(* Logix 5000 project; controller ABB_Drive_Test vendor 1 type 14 code 151 rev 33.13; software revision 33.01 *)

TASK MainTask (continuous, watchdog 500 ms) : T000_MainProgram

MODULES
   Local : vendor 1 type 14 code 151 (Compact 0, rev 33.13)
      Analog_IO : Embedded (Compact 2, rev 1.1, Output RPI 80 ms)
      Module_Hart : vendor 58 type 10 code 4 (Compact 4, rev 3.1, Output RPI 80 ms)
      Discrete_IO : Embedded (Compact 1, rev 3.1, Output RPI 20 ms)
      Counters : Embedded (Compact 3, rev 1.1, Output RPI 20 ms)
      PLC : 1769-L32E Ethernet Port (Ethernet 192.168.2.131, rev 20.1)
         PLC_Controller : vendor 1 type 14 code 77 (CompactLogixL32EController 0, rev 20.1, $7a3aac4c$ RPI 20 ms, $3ca1aa1f$ RPI 20 ms, $2d7d331d$ RPI 20 ms)
      ABBDrive : ETHERNET-MODULE (Ethernet 192.168.2.9, rev 1.1, Output RPI 20 ms)
           ABBDrive:I.Data[0]   // Logic Status Word
           ABBDrive:I.Data[1]   // RPM Actual (INT)
           ABBDrive:I.Data[2]   // DL 1 (Real)
           ABBDrive:I.Data[3]   // DL 1 (Real)
END_MODULES

TYPE ABB_Read :   // Datalinks de Lectura
STRUCT
   Logic_Status_Word : LSW;
   RPM_Feedback : INT;   // RPM Tomada del VSD
   RPM_Referencia : INT;   // Referencia RPM Inyectada
   Output_Power : REAL;
   BusDC : REAL;
   Output_Current : REAL;
   Output_Voltage : REAL;
   PF : REAL;   // Factor de Potencia
   Latest_Fault : INT;
   Accel : BOOL;   // Estado VSD si esta Acelerando
   Descell : BOOL;   // Estado VSD si esta Deshacelerando
END_STRUCT
END_TYPE

TYPE ABB_Write :
STRUCT
   RPM_Reference : INT;
   Run_Forward : BOOL;
   Run_Reverse : BOOL;
   Reset_Fault : BOOL;
END_STRUCT
END_TYPE

TYPE ComandVSD :   // Comandos de funcionamiento VSD
STRUCT
   start : BOOL;   // arranque
   stop : BOOL;   // Parada
   reset : BOOL;   // reset VSD
   referencia : REAL;   // Referencia en RPM para VSD AFE
   direction : BOOL;   // Fordware o Reverse
END_STRUCT
END_TYPE

TYPE Dinagrama :   // Estructura para el dinagrama
STRUCT
   vPotencia : REAL[500];   // captura del vector de potencia
   vCarga : REAL[500];   // captura del vector de carga
   vPosicion : REAL[500];   // captura del vector posicion
   vProximetro : DINT[500];   // captura del vector del proximetro
   NumeroMuestras : INT;
   enabled : BOOL;
   captura : BOOL;   // Flag que indica la captura del sistema
   resetVector : BOOL;   // Flag para darle Reset al vector de posición y carga
   vEmptyREAL : REAL[500];
   vEmptyINT : DINT[500];
   tMuestreo : REAL;   // Tiempo de Muestreo de captura
END_STRUCT
END_TYPE

TYPE ethImplicitRead :   // Comunicación para la lectura de los parametros del VSD por ethernet IP
STRUCT
   Enabled : BOOL;   // habilitar Comunicación
   Done : BOOL;   // Se realizó correctamente
   Error : BOOL;   // Se tiene un error en la lectura de los parámetros
   Value : DINT;   // Valor Obtenido
   instance : DINT;   // instancia del parametro
   atribute : INT;   // Atributo del parametro
END_STRUCT
END_TYPE

TYPE ethImplicitWrite :   // Comunicación Para enviar parametros al sistema
STRUCT
   Enabled : BOOL;   // Habilitar
   Done : BOOL;   // Se realizo exitozamente
   ERR : BOOL;   // Error en el envio de la información
   Value : DINT;   // Valor a ingresar
   Instance : DINT;   // Valor de la Instancia
   Atribute : INT;   // Valor del Atributo de la instancia
   clase : INT;
END_STRUCT
END_TYPE

TYPE fuenteEntradaAnaloga :   // Definición de Entrada Analoga ,Fuente de la señal ,rango minimo y maximo
STRUCT
   fuente : INT;   // Canal por el cual se suministra la señal
   Valor : REAL;   // Valor Actual de la señal
   min : REAL;
   max : REAL;
   ValorMinAmp : REAL;
END_STRUCT
END_TYPE

TYPE LSW :   // Drive - Logic Status Word
STRUCT
   Faulted : BOOL;
   Warning : BOOL;
   RunForward : BOOL;
   RunReverse : BOOL;
   Ready : BOOL;
   RemoteRef : BOOL;
   RemoteCrtl : BOOL;
   AtSpeed : BOOL;
END_STRUCT
END_TYPE

TYPE SWC :   // Comunicación Ethernet con el SWC PRO
STRUCT
   comand : ComandVSD;   // Comandos para VSD
   Dinagrama : Dinagrama;   // Valores para adquisión del dinagrama
   entradasDigitales : INT;
   salidasDigitales : INT;
   entradasAnalogas : REAL[4];
   salidasAnalogas : REAL[4];
   ABBRead : ABB_Read;   // Valores de Lectura
   etheWrite : ethImplicitWrite;   // Valores de Escritura Ethernet para VSD
   etheRead : ethImplicitRead;   // Valores de Lectura
END_STRUCT
END_TYPE

VAR_GLOBAL   (* controller tags *)
   ABB_GetAtt_Value : DINT := 6000;
   ABB_GetMsg : MESSAGE;
        MessageParameters(ServiceCode := 16#000e, DestinationTag := ABB_GetAtt_Value, ...)
   ABB_Input : ABB_Read := (Logic_Status_Word.Ready := 1, Logic_Status_Word.RemoteRef := 1, Logic_Status_Word.RemoteCrtl := 1, RPM_Referencia := 72, Output_Power := 5.960401e-37, BusDC := 715.4, PF := 1.0, Latest_Fault := 28801);
   ABB_Msg_SetValue : DINT := 1;
   ABB_Output : ABB_Write := (RPM_Reference := 72);
   ABB_SetMsg : MESSAGE;
        MessageParameters(ServiceCode := 16#0010, LocalElement := ABB_Msg_SetValue, ...)
   counters : COUNTER[20];
        [0]   // C indice Dinagrama
   Proximetro : BOOL;
   SRP_Displacement_Actual : REAL := 11.377348;
   SRP_Load_Actual : REAL := 10.545264;
   SRP_SimActualStroke : DINT;
   SWC : SWC := (comand.referencia := 72.0, comand.direction := 1, Dinagrama.tMuestreo := 0.05, entradasAnalogas[0] := 16.901644, entradasAnalogas[1] := 13.587194, entradasAnalogas[2] := 3.2056525, entradasAnalogas[3] := 3.2056525, ABBRead.Logic_Status_Word.Ready := 1, ABBRead.Logic_Status_Word.RemoteRef := 1, ABBRead.Logic_Status_Word.RemoteCrtl := 1, ABBRead.RPM_Referencia := 72, ABBRead.Output_Power := 5.960401e-37, ABBRead.BusDC := 714.3, ABBRead.PF := 1.0, ABBRead.Latest_Fault := 28801, etheWrite.Value := 1, etheWrite.Instance := 99, etheWrite.Atribute := 13, etheRead.Value := 6000, etheRead.instance := 99, etheRead.atribute := 7);
   Timmers : TIMER[10] := ([0].PRE := 43, [1].PRE := 828000, [1].ACC := 352537, [1].EN := 1, [1].TT := 1, [2].PRE := 500, [3].PRE := 200, [4].PRE := 10000);
        [0]   // tMuestreo
        [1]   // tPausa
        [2]   // reset del done write ethet
        [3]   // reset del done read eth
        [4]   // reset de la flag de arranque
END_VAR

PROGRAM T000_MainProgram   (* main routine R00_MainRoutine *)
VAR
   Acell : BOOL;
   Captura : BOOL := 1;
   contadorAux : ALIAS FOR counter[0].ACC;
   counter : COUNTER[10] := ([0].DN := 1);
   DesAcell : BOOL;
   Flag : BOOL;
   flagDesAcell : BOOL;   // Flag Auxiliar Boton de Parada
   indiceLocal : DINT;
   InicioDinagram : BOOL := 1;   // Inicio de la Adquisión del Dinagrama
   myoneshot : BOOL[32];
        [0]   // oneshot toogle bot dinagrama
        [2]   // reset de la flag cuando se habilita y se deshabilita
        [1]   // oneshor reset del ocntador
   numeroMuestras : DINT := 640;   // Numero de Muestras del Stroke
   pausa : BOOL := 1;
   Proximetro_Virtual : ALIAS FOR SRP_SimActualStroke;
   rpmFeedback : INT;   // Valor absoluto de la referencia 0 no lo toma
   SCL_01 : SCALE := (In := 16890.0, InRawMax := 19987.0, InRawMin := 3994.0, InEUMax := 20.0, InEUMin := 4.0, Out := 16.901644);
   SCL_02 : SCALE := (In := 13577.0, InRawMax := 19987.0, InRawMin := 3994.0, InEUMax := 20.0, InEUMin := 4.0, Out := 13.587194);
   SCL_03 : SCALE := (In := 3200.0, InRawMax := 19987.0, InRawMin := 3994.0, InEUMax := 20.0, InEUMin := 4.0, Out := 3.2056525, MinAlarm := 1);
   SCL_04 : SCALE := (In := 3200.0, InRawMax := 19987.0, InRawMin := 3994.0, InEUMax := 20.0, InEUMin := 4.0, Out := 3.2056525, MinAlarm := 1);
   SPM_Reference : REAL := 8.5;
   timer : TIMER[10] := ([0].PRE := 50);
        [0]   // Tiempo Muestreo
   VCarga : REAL[1500] := ([0] := 11.827799, [1] := 8.980304, [2] := 8.936409, [3] := 8.84487, [4] := 8.84487, [5] := 8.963797, [6] := 8.963797, [7] := 8.966047, [8] := 8.966047, [9] := 8.860626, [10] := 8.860626, [11] := 9.400863, [12] := 9.400863, [13] := 9.521291, [14] := 9.4916525, [15] := 9.4916525, [16] := 9.597824, [17] := 9.597824, [18] := 9.593322, [19] := 9.593322, [20] := 9.387732, [21] := 9.387732, [22] := 9.403114, [23] := 9.403114, [24] := 9.185143, [25] := 9.185143, [26] := 8.987057, [27] := 8.668918, [28] := 8.668918, [29] := 8.395048, [30] := 8.395048, [31] := 7.648096, [32] := 7.648096, [33] := 7.4162445, [34] := 7.4162445, [35] := 7.2624273, [36] := 7.2624273, [37] := 6.939786, [38] := 6.784468, [39] := 6.784468, [40] := 6.619771, [41] := 6.619771, [42] := 6.1519413, [43] := 6.1519413, [44] := 6.0791597, [45] := 6.0791597, [46] := 6.3091354, [47] := 6.3091354, [48] := 6.480585, [49] := 6.480585, [50] := 6.990058, [51] := 7.45151, [52] := 7.45151, [53] := 7.4702682, [54] := 7.4702682, [55] := 7.577565, [56] := 7.577565, [57] := 7.7895327, [58] := 7.7895327, [59] := 7.948227,
        [60] := 7.948227, [61] := 8.027012, [62] := 8.353029, [63] := 8.353029, [64] := 8.441193, [65] := 8.441193, [66] := 8.438942, [67] := 8.438942, [68] := 8.222097, [69] := 8.222097, [70] := 8.014256, [71] := 8.014256, [72] := 8.062653, [73] := 8.062653, [74] := 8.050648, [75] := 8.092665, [76] := 8.092665, [77] := 8.186457, [78] := 8.186457, [79] := 8.133558, [80] := 8.133558, [81] := 8.182329, [82] := 8.182329, [83] := 8.211593, [84] := 8.211593, [85] := 8.28625, [86] := 8.660664, [87] := 8.660664, [88] := 8.850497, [89] := 8.850497, [90] := 9.020447, [91] := 9.020447, [92] := 9.068843, [93] := 9.068843, [94] := 9.367474, [95] := 9.367474, [96] := 9.479647, [97] := 9.479647, [98] := 9.492778, [99] := 9.546427, [100] := 9.546427, [101] := 9.607578, [102] := 9.607578, [103] := 9.483774, [104] := 9.483774, [105] := 9.460889, [106] := 9.460889, [107] := 9.368223, [108] := 9.368223, [109] := 9.679609, [110] := 10.03639, [111] := 10.03639, [112] := 10.411555, [113] := 10.411555, [114] := 10.760458, [115] := 10.760458, [116] := 10.886138, [117] := 10.886138, [118] := 11.210654, [119] := 11.210654,
        [120] := 11.363346, [121] := 11.575314, [122] := 11.575314, [123] := 11.714874, [124] := 11.714874, [125] := 11.875445, [126] := 11.875445, [127] := 11.921966, [128] := 11.921966, [129] := 11.762521, [130] := 11.762521, [131] := 11.252673, [132] := 11.252673, [133] := 11.074845, [134] := 10.70906, [135] := 10.70906, [136] := 10.527856, [137] := 10.527856, [138] := 10.288126, [139] := 10.288126, [140] := 10.021759, [141] := 10.021759, [142] := 9.853685, [143] := 9.853685, [144] := 9.544551, [145] := 9.442506, [146] := 9.442506, [147] := 9.472519, [148] := 9.472519, [149] := 9.855186, [150] := 9.855186, [151] := 9.900206, [152] := 9.900206, [153] := 10.149315, [154] := 10.149315, [155] := 10.241606, [156] := 10.265241, [157] := 10.265241, [158] := 10.363909, [159] := 10.363909, [160] := 10.395048, [161] := 10.395048, [162] := 10.3444, [163] := 10.3444, [164] := 10.475332, [165] := 10.475332, [166] := 10.469706, [167] := 10.469706, [168] := 10.228475, [169] := 9.813543, [170] := 9.813543, [171] := 9.537798, [172] := 9.537798, [173] := 9.315701, [174] := 9.315701, [175] := 9.132996, [176] := 9.132996, [177] := 9.119114, [178] := 9.119114, [179] := 8.870006,
        [180] := 8.735697, [181] := 8.735697, [182] := 8.758582, [183] := 8.758582, [184] := 8.534609, [185] := 8.534609, [186] := 8.67642, [187] := 8.67642, [188] := 9.151003, [189] := 9.151003, [190] := 9.39336, [191] := 9.39336, [192] := 9.578316, [193] := 9.796661, [194] := 9.796661, [195] := 9.773776, [196] := 9.773776, [197] := 9.757269, [198] := 9.757269, [199] := 9.786156, [200] := 9.786156, [201] := 9.807541, [202] := 9.807541, [203] := 9.934346, [204] := 9.906584, [205] := 9.906584, [206] := 9.544926, [207] := 9.544926, [208] := 9.334833, [209] := 9.334833, [210] := 9.290565, [211] := 9.290565, [212] := 9.1633835, [213] := 9.1633835, [214] := 8.979178, [215] := 9.039205, [216] := 9.039205, [217] := 8.922528, [218] := 8.922528, [219] := 8.92628, [220] := 8.92628, [221] := 8.94879, [222] := 8.94879, [223] := 8.869631, [224] := 8.869631, [225] := 9.230538, [226] := 9.230538, [227] := 9.474395, [228] := 9.451135, [229] := 9.451135, [230] := 9.526167, [231] := 9.526167, [232] := 9.65785, [233] := 9.65785, [234] := 9.437254, [235] := 9.437254, [236] := 9.396736, [237] := 9.396736, [238] := 9.276684, [239] := 9.276684,
        [240] := 9.073344, [241] := 8.794222, [242] := 8.794222, [243] := 8.592009, [244] := 8.592009, [245] := 7.9212155, [246] := 7.9212155, [247] := 7.471769, [248] := 7.471769, [249] := 7.410617, [250] := 7.410617, [251] := 7.0429564, [252] := 6.733821, [253] := 6.733821, [254] := 6.701932, [255] := 6.701932, [256] := 6.272744, [257] := 6.272744, [258] := 6.0765333, [259] := 6.0765333, [260] := 6.197336, [261] := 6.197336, [262] := 6.3331456, [263] := 6.6576624, [264] := 6.6576624, [265] := 6.9412866, [266] := 6.9412866, [267] := 7.467267, [268] := 7.467267, [269] := 7.4646406, [270] := 7.4646406, [271] := 7.641343, [272] := 7.641343, [273] := 7.919339, [274] := 7.919339, [275] := 7.933221, [276] := 8.245732, [277] := 8.245732, [278] := 8.452448, [279] := 8.452448, [280] := 8.443819, [281] := 8.443819, [282] := 8.419058, [283] := 8.419058, [284] := 8.013506, [285] := 8.013506, [286] := 8.006377, [287] := 8.051773, [288] := 8.051773, [289] := 8.016132, [290] := 8.016132, [291] := 8.186081, [292] := 8.186081, [293] := 8.177452, [294] := 8.177452, [295] := 8.110298, [296] := 8.110298, [297] := 8.171075, [298] := 8.210467, [299] := 8.210467,
        [300] := 8.3988, [301] := 8.3988, [302] := 8.589007, [303] := 8.589007, [304] := 8.928906, [305] := 8.928906, [306] := 9.02795, [307] := 9.02795, [308] := 9.220784, [309] := 9.419996, [310] := 9.419996, [311] := 9.439505, [312] := 9.439505, [313] := 9.462765, [314] := 9.462765, [315] := 9.537047, [316] := 9.537047, [317] := 9.573063, [318] := 9.573063, [319] := 9.490152, [320] := 9.4698925, [321] := 9.4698925, [322] := 9.459013, [323] := 9.459013, [324] := 9.643969, [325] := 9.643969, [326] := 10.221722, [327] := 10.221722, [328] := 10.381166, [329] := 10.381166, [330] := 10.706809, [331] := 10.706809, [332] := 11.081974, [333] := 11.236916, [334] := 11.236916, [335] := 11.451885, [336] := 11.451885, [337] := 11.557682, [338] := 11.557682, [339] := 11.815419, [340] := 11.815419, [341] := 11.894579, [342] := 11.894579, [343] := 11.83943, [344] := 11.502533, [345] := 11.502533, [346] := 11.23354, [347] := 11.23354, [348] := 10.874508, [349] := 10.874508, [350] := 10.510599, [351] := 10.510599, [352] := 10.356781, [353] := 10.356781, [354] := 10.096416, [355] := 10.096416, [356] := 9.954229, [357] := 9.64622, [358] := 9.64622, [359] := 9.505158,
        [360] := 9.505158, [361] := 9.400863, [362] := 9.400863, [363] := 9.780153, [364] := 9.780153, [365] := 9.882948, [366] := 9.882948, [367] := 10.071281, [368] := 10.19546, [369] := 10.19546, [370] := 10.254736, [371] := 10.254736, [372] := 10.277621, [373] := 10.277621, [374] := 10.384542, [375] := 10.384542, [376] := 10.339899, [377] := 10.339899, [378] := 10.465578, [379] := 10.506472, [380] := 10.506472, [381] := 10.054024, [382] := 10.054024, [383] := 9.839805, [384] := 9.839805, [385] := 9.606077, [386] := 9.606077, [387] := 9.399737, [388] := 9.399737, [389] := 9.1281185, [390] := 9.1281185, [391] := 9.126243, [392] := 8.908272, [393] := 8.908272, [394] := 8.755205, [395] := 8.755205, [396] := 8.7780905, [397] := 8.7780905, [398] := 8.501595, [399] := 8.501595, [400] := 8.5837555, [401] := 8.5837555, [402] := 9.026824, [403] := 9.205777, [404] := 9.205777, [405] := 9.39636, [406] := 9.39636, [407] := 9.727256, [408] := 9.727256, [409] := 9.79591, [410] := 9.79591, [411] := 9.780529, [412] := 9.780529, [413] := 9.807541, [414] := 9.807541, [415] := 9.803789, [416] := 9.897205, [417] := 9.897205, [418] := 9.930969, [419] := 9.930969,
        [420] := 9.623335, [421] := 9.623335, [422] := 9.400488, [423] := 9.400488, [424] := 9.295442, [425] := 9.295442, [426] := 9.008066, [427] := 8.962296, [428] := 8.962296, [429] := 9.047083, [430] := 9.047083, [431] := 8.975801, [432] := 8.975801, [433] := 8.909022, [434] := 8.909022, [435] := 8.966047, [436] := 8.966047, [437] := 8.890639, [438] := 9.06209, [439] := 9.06209, [440] := 9.338211, [441] := 9.338211, [442] := 9.465767, [443] := 9.465767, [444] := 9.556181, [445] := 9.556181, [446] := 9.638342, [447] := 9.638342, [448] := 9.448133, [449] := 9.448133, [450] := 9.385857, [451] := 9.296942, [452] := 9.296942, [453] := 9.101857, [454] := 9.101857, [455] := 8.818608, [456] := 8.818608, [457] := 8.357906, [458] := 8.357906, [459] := 7.983493, [460] := 7.983493, [461] := 7.4822736, [462] := 7.410617, [463] := 7.410617, [464] := 7.021572, [465] := 7.021572, [466] := 6.8223596, [467] := 6.8223596, [468] := 6.7008066, [469] := 6.7008066, [470] := 6.2479835, [471] := 6.2479835, [472] := 6.0566497, [473] := 6.0566497, [474] := 6.2190957, [475] := 6.393172, [476] := 6.393172, [477] := 6.8107295, [478] := 6.8107295, [479] := 7.374226,
        [480] := 7.374226, [481] := 7.45076, [482] := 7.45076, [483] := 7.5531793, [484] := 7.5531793, [485] := 7.767773, [486] := 7.942975, [487] := 7.942975, [488] := 8.143312, [489] := 8.143312, [490] := 8.344026, [491] := 8.344026, [492] := 8.444944, [493] := 8.444944, [494] := 8.4396925, [495] := 8.4396925, [496] := 8.304258, [497] := 8.096416, [498] := 8.096416, [499] := 8.028888, [500] := 8.028888, [501] := 8.033765, [502] := 8.033765, [503] := 8.07991, [504] := 8.07991, [505] := 8.186457, [506] := 8.186457, [507] := 8.135059, [508] := 8.135059, [509] := 8.197711, [510] := 8.211593, [511] := 8.211593, [512] := 8.229976, [513] := 8.229976, [514] := 8.545488, [515] := 8.545488, [516] := 8.742825, [517] := 8.742825, [518] := 8.9941845, [519] := 8.9941845, [520] := 9.020071, [521] := 9.285313, [522] := 9.285313, [523] := 9.451509, [524] := 9.451509, [525] := 9.517163, [526] := 9.517163, [527] := 9.464266, [528] := 9.464266, [529] := 9.501032, [530] := 9.501032, [531] := 9.53367, [532] := 9.502157, [533] := 9.502157, [534] := 9.4275, [535] := 9.4275, [536] := 9.529919, [537] := 9.529919, [538] := 9.845057, [539] := 9.845057,
        [540] := 10.316263, [541] := 10.316263, [542] := 10.42281, [543] := 10.777716, [544] := 10.777716, [545] := 11.084224, [546] := 11.084224, [547] := 11.248171, [548] := 11.248171, [549] := 11.445131, [550] := 11.445131, [551] := 11.532545, [552] := 11.532545, [553] := 11.782029, [554] := 11.782029, [555] := 11.825172, [556] := 11.940723, [557] := 11.940723, [558] := 11.577189, [559] := 11.577189, [560] := 11.331833, [561] := 11.331833, [562] := 10.911648, [563] := 10.911648, [564] := 10.58338, [565] := 10.58338, [566] := 10.444944, [567] := 10.190208, [568] := 10.190208, [569] := 10.078409, [570] := 10.078409, [571] := 9.809792, [572] := 9.809792, [573] := 9.529544, [574] := 9.529544, [575] := 9.457888, [576] := 9.457888, [577] := 9.594072, [578] := 9.594072, [579] := 9.784656, [580] := 9.956106, [581] := 9.956106, [582] := 10.071656, [583] := 10.071656, [584] := 10.249859, [585] := 10.249859, [586] := 10.2806225, [587] := 10.2806225, [588] := 10.339523, [589] := 10.339523, [590] := 10.348528, [591] := 10.3391485, [592] := 10.3391485, [593] := 10.590883, [594] := 10.590883, [595] := 10.506846, [596] := 10.506846, [597] := 10.029263, [598] := 10.029263, [599] := 9.728756,
        [600] := 9.728756, [601] := 9.62221, [602] := 9.1933975, [603] := 9.1933975, [604] := 9.127743, [605] := 9.127743, [606] := 9.046708, [607] := 9.046708, [608] := 8.771712, [609] := 8.771712, [610] := 8.722941, [611] := 8.722941, [612] := 8.703433, [613] := 8.556744, [614] := 8.556744, [615] := 8.787845, [616] := 8.787845, [617] := 9.044832, [618] := 9.044832, [619] := 9.310448, [620] := 9.310448, [621] := 9.667979, [622] := 9.667979, [623] := 9.759895, [624] := 9.779028, [625] := 9.779028, [626] := 9.782405, [627] := 9.782405, [628] := 9.8082905, [629] := 9.8082905, [630] := 9.803413, [631] := 9.803413, [632] := 9.923091, [633] := 9.923091, [634] := 9.797411, [635] := 9.345714, [636] := 9.345714, [637] := 9.306322, [638] := 9.306322, [639] := 9.172388, [640] := 9.172388, [641] := 11.520915, [642] := 11.266179, [643] := 10.959294, [644] := 10.632902, [645] := 10.337273, [646] := 9.96511, [647] := 9.549427, [648] := 9.102608, [649] := 8.607766, [650] := 8.366911, [651] := 7.9463515, [652] := 7.4500093, [653] := 7.020071, [654] := 6.6572876, [655] := 6.3882947, [656] := 6.1879573, [657] := 6.123429, [658] := 6.1515665, [659] := 6.306509,
        [660] := 6.5207276, [661] := 6.867755, [662] := 7.260176, [663] := 7.6889887, [664] := 8.14819, [665] := 8.538361, [666] := 9.081598, [667] := 9.579441, [668] := 10.054773, [669] := 10.433314, [670] := 10.879759, [671] := 11.271807, [672] := 11.602701, [673] := 11.830425, [674] := 11.960233, [675] := 12.053648, [676] := 12.062277, [677] := 11.9992485, [678] := 11.901332, [679] := 11.737385, [680] := 11.539298, [681] := 11.306321, [682] := 11.069968, [683] := 10.769087, [684] := 10.393923, [685] := 10.046896, [686] := 9.717501, [687] := 9.266179, [688] := 8.839993, [689] := 8.358657, [690] := 7.861564, [691] := 7.5719376, [692] := 7.1783905, [693] := 6.7642093, [694] := 6.470831, [695] := 6.2318516, [696] := 6.1268053, [697] := 6.1283064, [698] := 6.2566123, [699] := 6.5015945, [700] := 6.829488, [701] := 7.2567997, [702] := 7.5719376, [703] := 8.032264, [704] := 8.511349, [705] := 8.931157, [706] := 9.431252, [707] := 9.95348, [708] := 10.449821, [709] := 10.877884, [710] := 11.1885195, [711] := 11.550178, [712] := 11.802288, [713] := 11.975239, [714] := 12.04577, [715] := 12.064903, [716] := 12.011254, [717] := 11.886701, [718] := 11.722754, [719] := 11.55468,
        [720] := 11.320202, [721] := 11.037329, [722] := 10.713187, [723] := 10.439317, [724] := 10.081785, [725] := 9.656725, [726] := 9.211781, [727] := 8.746576, [728] := 8.394298, [729] := 7.8938284, [730] := 7.385481, [731] := 7.0384545, [732] := 6.6576624, [733] := 6.37704, [734] := 6.25061, [735] := 6.135434, [736] := 6.132808, [737] := 6.2322264, [738] := 6.4569497, [739] := 6.781467, [740] := 7.156631, [741] := 7.580191, [742] := 7.9636087, [743] := 8.440818, [744] := 8.94879, [745] := 9.467642, [746] := 9.989495, [747] := 10.374788, [748] := 10.827987, [749] := 11.235415, [750] := 11.583942, [751] := 11.786907, [752] := 11.959857, [753] := 12.050648, [754] := 12.062277, [755] := 12.019883, [756] := 11.9020815, [757] := 11.734009, [758] := 11.524292, [759] := 11.287188, [760] := 11.042206, [761] := 10.725567, [762] := 10.368411, [763] := 9.978615, [764] := 9.63459, [765] := 9.160382, [766] := 8.693303, [767] := 8.187207, [768] := 7.703245, [769] := 7.3678484, [770] := 6.9619207, [771] := 6.610392, [772] := 6.3822923, [773] := 6.1935844, [774] := 6.1204276, [775] := 6.166948, [776] := 6.2453575, [777] := 6.5045958, [778] := 6.717689, [779] := 7.077096,
        [780] := 7.525042, [781] := 7.968111, [782] := 8.438566, [783] := 8.844494, [784] := 9.386982, [785] := 9.897205, [786] := 10.383793, [787] := 10.742825, [788] := 11.151003, [789] := 11.49878, [790] := 11.775652, [791] := 11.959482, [792] := 12.040893, [793] := 12.066403, [794] := 12.021384, [795] := 11.910336, [796] := 11.785781, [797] := 11.588445, [798] := 11.33746, [799] := 11.060964, [800] := 11.060964);
   VPosicion : REAL[1500] := ([0] := 97.12999, [1] := 94.7602, [2] := 93.322075, [3] := 92.56549, [4] := 92.56549, [5] := 91.0961, [6] := 91.0961, [7] := 90.23948, [8] := 90.23948, [9] := 88.451195, [10] := 88.451195, [11] := 86.787964, [12] := 86.787964, [13] := 85.76877, [14] := 83.62408, [15] := 83.62408, [16] := 82.62365, [17] := 82.62365, [18] := 80.466446, [19] := 80.466446, [20] := 78.15294, [21] := 78.15294, [22] := 76.933655, [23] := 76.933655, [24] := 74.39504, [25] := 74.39504, [26] := 73.175766, [27] := 70.61214, [28] := 70.61214, [29] := 69.317825, [30] := 69.317825, [31] := 66.622894, [32] := 66.622894, [33] := 63.784153, [34] := 63.784153, [35] := 62.489838, [36] := 62.489838, [37] := 59.6636, [38] := 58.469326, [39] := 58.469326, [40] := 55.436752, [41] := 55.436752, [42] := 52.37916, [43] := 52.37916, [44] := 50.815983, [45] := 50.815983, [46] := 47.683357, [47] := 47.683357, [48] := 46.12018, [49] := 46.12018, [50] := 42.912518, [51] := 39.686108, [52] := 39.686108, [53] := 38.079155, [54] := 38.079155, [55] := 33.921085, [56] := 33.921085, [57] := 32.795597, [58] := 32.795597, [59] := 30.0569,
        [60] := 30.0569, [61] := 26.43031, [62] := 25.311077, [63] := 25.311077, [64] := 22.603638, [65] := 22.603638, [66] := 20.752829, [67] := 20.752829, [68] := 18.23923, [69] := 18.23923, [70] := 16.82611, [71] := 16.82611, [72] := 14.187455, [73] := 14.187455, [74] := 11.79266, [75] := 10.367036, [76] := 10.367036, [77] := 8.122304, [78] := 8.122304, [79] := 6.3465266, [80] := 6.3465266, [81] := 5.589944, [82] := 5.589944, [83] := 4.3706627, [84] := 4.3706627, [85] := 3.826675, [86] := 2.901268, [87] := 2.901268, [88] := 2.5573702, [89] := 2.5573702, [90] := 2.1071732, [91] := 2.1071732, [92] := 2.0008743, [93] := 2.0008743, [94] := 2.0008743, [95] := 2.0008743, [96] := 2.4073033, [97] := 2.4073033, [98] := 2.6949286, [99] := 3.532797, [100] := 3.532797, [101] := 4.0892897, [102] := 4.0892897, [103] := 5.277309, [104] := 5.277309, [105] := 6.9655476, [106] := 6.9655476, [107] := 7.9159617, [108] := 7.9159617, [109] := 9.666729, [110] := 10.861, [111] := 10.861, [112] := 13.07447, [113] := 13.07447, [114] := 15.544301, [115] := 15.544301, [116] := 16.813606, [117] := 16.813606, [118] := 19.714874, [119] := 19.714874,
        [120] := 22.459826, [121] := 23.829174, [122] := 23.829174, [123] := 26.699179, [124] := 26.699179, [125] := 28.068531, [126] := 28.068531, [127] := 31.263674, [128] := 31.263674, [129] := 32.514225, [130] := 32.514225, [131] := 35.302944, [132] := 35.302944, [133] := 38.954544, [134] := 40.624023, [135] := 40.624023, [136] := 43.6566, [137] := 43.6566, [138] := 45.588696, [139] := 45.588696, [140] := 49.415367, [141] := 49.415367, [142] := 51.247417, [143] := 51.247417, [144] := 54.798973, [145] := 57.769024, [146] := 57.769024, [147] := 59.476017, [148] := 59.476017, [149] := 63.05258, [150] := 63.05258, [151] := 66.10392, [152] := 66.10392, [153] := 67.83593, [154] := 67.83593, [155] := 71.32495, [156] := 72.938156, [157] := 72.938156, [158] := 76.15831, [159] := 76.15831, [160] := 77.32133, [161] := 77.32133, [162] := 79.92871, [163] := 79.92871, [164] := 82.8675, [165] := 82.8675, [166] := 84.33064, [167] := 84.33064, [168] := 86.79422, [169] := 87.750885, [170] := 87.750885, [171] := 90.14568, [172] := 90.14568, [173] := 91.15238, [174] := 91.15238, [175] := 93.28456, [176] := 93.28456, [177] := 94.95404, [178] := 94.95404, [179] := 95.823166,
        [180] := 97.292564, [181] := 97.292564, [182] := 97.93659, [183] := 97.93659, [184] := 99.10586, [185] := 99.10586, [186] := 99.98748, [187] := 99.98748, [188] := 100.35015, [189] := 100.35015, [190] := 100.831604, [191] := 100.831604, [192] := 101.10673, [193] := 101.1505, [194] := 101.1505, [195] := 101.07547, [196] := 101.07547, [197] := 100.981674, [198] := 100.981674, [199] := 100.66904, [200] := 100.66904, [201] := 100.43769, [202] := 100.43769, [203] := 99.80617, [204] := 99.11211, [205] := 99.11211, [206] := 98.79322, [207] := 98.79322, [208] := 97.78027, [209] := 97.78027, [210] := 97.2613, [211] := 97.2613, [212] := 96.16706, [213] := 96.16706, [214] := 95.5293, [215] := 94.08491, [216] := 94.08491, [217] := 92.65304, [218] := 92.65304, [219] := 91.77765, [220] := 91.77765, [221] := 90.38329, [222] := 90.38329, [223] := 88.33864, [224] := 88.33864, [225] := 87.469505, [226] := 87.469505, [227] := 85.599945, [228] := 84.59325, [229] := 84.59325, [230] := 82.56111, [231] := 82.56111, [232] := 81.46689, [233] := 81.46689, [234] := 79.20339, [235] := 79.20339, [236] := 76.72732, [237] := 76.72732, [238] := 75.73938, [239] := 75.73938,
        [240] := 73.12574, [241] := 71.85643, [242] := 71.85643, [243] := 69.22404, [244] := 69.22404, [245] := 67.92346, [246] := 67.92346, [247] := 65.19727, [248] := 65.19727, [249] := 62.63365, [250] := 62.63365, [251] := 61.23929, [252] := 58.519352, [253] := 58.519352, [254] := 55.29294, [255] := 55.29294, [256] := 53.81729, [257] := 53.81729, [258] := 50.60339, [259] := 50.60339, [260] := 49.040203, [261] := 49.040203, [262] := 46.74545, [263] := 43.431496, [264] := 43.431496, [265] := 41.937096, [266] := 41.937096, [267] := 38.37304, [268] := 38.37304, [269] := 36.722313, [270] := 36.722313, [271] := 33.46464, [272] := 33.46464, [273] := 31.776405, [274] := 31.776405, [275] := 28.518724, [276] := 26.223969, [277] := 26.223969, [278] := 24.592007, [279] := 24.592007, [280] := 21.57819, [281] := 21.57819, [282] := 18.733194, [283] := 18.733194, [284] := 17.001188, [285] := 17.001188, [286] := 14.350027, [287] := 13.080722, [288] := 13.080722, [289] := 10.773462, [290] := 10.773462, [291] := 9.879321, [292] := 9.879321, [293] := 7.965985, [294] := 7.965985, [295] := 6.3340216, [296] := 6.3340216, [297] := 5.5149136, [298] := 4.2268486, [299] := 4.2268486,
        [300] := 3.61408, [301] := 3.61408, [302] := 2.794972, [303] := 2.794972, [304] := 2.4760842, [305] := 2.4760842, [306] := 2.0634027, [307] := 2.0634027, [308] := 2.0008743, [309] := 2.0008743, [310] := 2.0008743, [311] := 2.4823368, [312] := 2.4823368, [313] := 3.2764344, [314] := 3.2764344, [315] := 3.695366, [316] := 3.695366, [317] := 4.945913, [318] := 4.945913, [319] := 5.6649776, [320] := 7.353216, [321] := 7.353216, [322] := 8.309886, [323] := 8.309886, [324] := 10.235727, [325] := 10.235727, [326] := 12.668043, [327] := 12.668043, [328] := 13.837301, [329] := 13.837301, [330] := 16.150814, [331] := 16.150814, [332] := 17.632713, [333] := 20.171326, [334] := 20.171326, [335] := 23.010067, [336] := 23.010067, [337] := 24.373161, [338] := 24.373161, [339] := 27.918465, [340] := 27.918465, [341] := 29.437876, [342] := 29.437876, [343] := 31.763899, [344] := 35.27168, [345] := 35.27168, [346] := 36.853622, [347] := 36.853622, [348] := 40.08629, [349] := 40.08629, [350] := 41.74951, [351] := 41.74951, [352] := 45.12599, [353] := 45.12599, [354] := 48.658787, [355] := 48.658787, [356] := 50.484585, [357] := 54.173695, [358] := 54.173695, [359] := 55.86194,
        [360] := 55.86194, [361] := 59.288437, [362] := 59.288437, [363] := 61.21428, [364] := 61.21428, [365] := 64.75958, [366] := 64.75958, [367] := 68.28612, [368] := 69.9431, [369] := 69.9431, [370] := 73.182014, [371] := 73.182014, [372] := 74.782715, [373] := 74.782715, [374] := 77.46514, [375] := 77.46514, [376] := 78.796974, [377] := 78.796974, [378] := 81.804535, [379] := 84.64328, [380] := 84.64328, [381] := 85.98762, [382] := 85.98762, [383] := 88.35115, [384] := 88.35115, [385] := 90.24573, [386] := 90.24573, [387] := 91.44626, [388] := 91.44626, [389] := 93.30332, [390] := 93.30332, [391] := 94.00987, [392] := 95.78565, [393] := 95.78565, [394] := 96.529724, [395] := 96.529724, [396] := 97.88657, [397] := 97.88657, [398] := 99.04332, [399] := 99.04332, [400] := 99.46226, [401] := 99.46226, [402] := 100.20634, [403] := 100.51272, [404] := 100.51272, [405] := 100.94416, [406] := 100.94416, [407] := 101.11298, [408] := 101.11298, [409] := 101.13174, [410] := 101.13174, [411] := 101.0317, [412] := 101.0317, [413] := 100.712814, [414] := 100.712814, [415] := 100.45644, [416] := 99.8937, [417] := 99.8937, [418] := 99.599815, [419] := 99.599815,
        [420] := 98.76821, [421] := 98.76821, [422] := 98.31801, [423] := 98.31801, [424] := 97.33007, [425] := 97.33007, [426] := 96.12956, [427] := 95.46051, [428] := 95.46051, [429] := 94.022385, [430] := 94.022385, [431] := 93.34083, [432] := 93.34083, [433] := 91.90271, [434] := 91.90271, [435] := 91.05233, [436] := 91.05233, [437] := 89.21403, [438] := 87.32571, [439] := 87.32571, [440] := 86.38153, [441] := 86.38153, [442] := 84.35565, [443] := 84.35565, [444] := 82.31726, [445] := 82.31726, [446] := 81.26055, [447] := 81.26055, [448] := 79.0846, [449] := 79.0846, [450] := 77.727745, [451] := 75.69561, [452] := 75.69561, [453] := 74.35753, [454] := 74.35753, [455] := 71.89395, [456] := 71.89395, [457] := 69.24279, [458] := 69.24279, [459] := 67.87344, [460] := 67.87344, [461] := 64.98468, [462] := 63.509033, [463] := 63.509033, [464] := 60.98918, [465] := 60.98918, [466] := 59.3197, [467] := 59.3197, [468] := 56.355904, [469] := 56.355904, [470] := 53.31082, [471] := 53.31082, [472] := 51.672607, [473] := 48.32114, [474] := 48.32114, [475] := 46.67667, [476] := 46.67667, [477] := 43.237663, [478] := 43.237663, [479] := 40.498966,
        [480] := 40.498966, [481] := 38.616898, [482] := 38.616898, [483] := 34.971546, [484] := 34.971546, [485] := 32.032764, [486] := 30.382038, [487] := 30.382038, [488] := 27.14312, [489] := 27.14312, [490] := 25.742508, [491] := 25.742508, [492] := 22.341024, [493] := 22.341024, [494] := 20.771587, [495] := 20.771587, [496] := 17.814043, [497] := 15.075344, [498] := 15.075344, [499] := 14.087415, [500] := 14.087415, [501] := 11.830175, [502] := 11.830175, [503] := 10.517102, [504] := 10.517102, [505] := 8.191085, [506] := 8.191085, [507] := 7.434502, [508] := 7.434502, [509] := 5.87132, [510] := 4.564497, [511] := 4.564497, [512] := 3.9454758, [513] := 3.9454758, [514] := 2.9763012, [515] := 2.9763012, [516] := 2.6198955, [517] := 2.6198955, [518] := 2.2072167, [519] := 2.2072167, [520] := 2.0071268, [521] := 2.0008743, [522] := 2.0008743, [523] := 2.1321833, [524] := 2.1321833, [525] := 2.7199388, [526] := 2.7199388, [527] := 3.101358, [528] := 3.101358, [529] := 4.0517716, [530] := 4.0517716, [531] := 4.8708797, [532] := 6.434065, [533] := 6.434065, [534] := 7.2844357, [535] := 7.2844357, [536] := 9.179014, [537] := 9.179014, [538] := 11.217406, [539] := 11.217406,
        [540] := 12.274119, [541] := 12.274119, [542] := 14.837742, [543] := 16.08829, [544] := 16.08829, [545] := 18.389297, [546] := 18.389297, [547] := 19.708622, [548] := 19.708622, [549] := 21.87832, [550] := 21.87832, [551] := 24.779589, [552] := 24.779589, [553] := 26.080154, [554] := 26.080154, [555] := 28.887642, [556] := 30.438316, [557] := 30.438316, [558] := 33.746017, [559] := 33.746017, [560] := 36.62852, [561] := 36.62852, [562] := 38.32927, [563] := 38.32927, [564] := 42.005875, [565] := 42.005875, [566] := 44.663284, [567] := 46.420307, [568] := 46.420307, [569] := 49.94685, [570] := 49.94685, [571] := 51.70387, [572] := 51.70387, [573] := 55.11161, [574] := 55.11161, [575] := 56.631023, [576] := 56.631023, [577] := 60.220093, [578] := 60.220093, [579] := 63.80291, [580] := 65.459885, [581] := 65.459885, [582] := 68.73007, [583] := 68.73007, [584] := 70.38704, [585] := 70.38704, [586] := 73.638466, [587] := 73.638466, [588] := 75.245415, [589] := 75.245415, [590] := 77.99661, [591] := 81.06672, [592] := 81.06672, [593] := 82.42355, [594] := 82.42355, [595] := 84.94341, [596] := 84.94341, [597] := 86.537865, [598] := 86.537865, [599] := 88.65753,
        [600] := 88.65753, [601] := 90.56462, [602] := 91.87144, [603] := 91.87144, [604] := 93.74726, [605] := 93.74726, [606] := 95.46676, [607] := 95.46676, [608] := 96.242096, [609] := 96.242096, [610] := 97.57394, [611] := 97.57394, [612] := 98.1617, [613] := 99.21841, [614] := 99.21841, [615] := 99.67486, [616] := 99.67486, [617] := 100.41892, [618] := 100.41892, [619] := 100.85663, [620] := 100.85663, [621] := 101.01295, [622] := 101.01295, [623] := 101.1505, [624] := 101.11298, [625] := 101.11298, [626] := 100.937904, [627] := 100.937904, [628] := 100.75658, [629] := 100.75658, [630] := 100.30013, [631] := 100.30013, [632] := 99.56231, [633] := 99.56231, [634] := 99.18089, [635] := 98.324265, [636] := 98.324265, [637] := 97.3676, [638] := 97.3676, [639] := 96.829865, [640] := 96.829865, [641] := 92.01525, [642] := 87.76965, [643] := 82.65491, [644] := 77.21503, [645] := 72.28787, [646] := 66.08516, [647] := 59.157127, [648] := 51.71012, [649] := 43.462765, [650] := 39.448513, [651] := 32.43919, [652] := 24.166822, [653] := 17.001188, [654] := 10.954791, [655] := 6.4715805, [656] := 3.1326203, [657] := 2.05715, [658] := 2.5261045, [659] := 5.1084847,
        [660] := 8.678797, [661] := 14.462578, [662] := 21.002937, [663] := 28.149813, [664] := 35.80316, [665] := 42.306007, [666] := 51.35997, [667] := 59.65735, [668] := 67.57956, [669] := 73.88857, [670] := 81.32932, [671] := 87.86345, [672] := 93.37836, [673] := 97.17376, [674] := 99.33721, [675] := 100.89414, [676] := 101.03796, [677] := 99.98748, [678] := 98.35553, [679] := 95.623085, [680] := 92.32163, [681] := 88.43869, [682] := 84.499466, [683] := 79.48477, [684] := 73.23204, [685] := 67.44826, [686] := 61.958355, [687] := 54.436314, [688] := 47.333206, [689] := 39.310944, [690] := 31.026072, [691] := 26.19896, [692] := 19.639843, [693] := 12.736821, [694] := 7.847184, [695] := 3.86419, [696] := 2.1134257, [697] := 2.1384358, [698] := 4.2768717, [699] := 8.359906, [700] := 13.824797, [701] := 20.946663, [702] := 26.19896, [703] := 33.871067, [704] := 41.855812, [705] := 48.852623, [706] := 57.187515, [707] := 65.89133, [708] := 74.1637, [709] := 81.298065, [710] := 86.47533, [711] := 92.50296, [712] := 96.7048, [713] := 99.58732, [714] := 100.76283, [715] := 101.08172, [716] := 100.18758, [717] := 98.11168, [718] := 95.379234, [719] := 92.578,
        [720] := 88.67004, [721] := 83.955475, [722] := 78.553116, [723] := 73.98862, [724] := 68.02976, [725] := 60.945408, [726] := 53.529667, [727] := 45.77627, [728] := 39.904957, [729] := 31.563807, [730] := 23.091352, [731] := 17.307573, [732] := 10.961044, [733] := 6.2839985, [734] := 4.1768284, [735] := 2.257237, [736] := 2.213469, [737] := 3.8704424, [738] := 7.6158314, [739] := 13.024449, [740] := 19.277185, [741] := 26.336521, [742] := 32.726814, [743] := 40.680294, [744] := 49.146496, [745] := 57.794033, [746] := 66.491585, [747] := 72.91315, [748] := 80.466446, [749] := 87.25692, [750] := 93.06571, [751] := 96.44845, [752] := 99.33095, [753] := 100.844124, [754] := 101.03796, [755] := 100.33139, [756] := 98.36803, [757] := 95.56681, [758] := 92.07153, [759] := 88.1198, [760] := 84.03676, [761] := 78.75945, [762] := 72.806854, [763] := 66.31026, [764] := 60.5765, [765] := 52.673042, [766] := 44.88839, [767] := 36.45345, [768] := 28.387415, [769] := 22.797472, [770] := 16.032013, [771] := 10.173202, [772] := 6.3715367, [773] := 3.2264113, [774] := 2.0071268, [775] := 2.782467, [776] := 4.0892897, [777] := 8.409929, [778] := 11.961484, [779] := 17.951601,
        [780] := 25.41737, [781] := 32.80185, [782] := 40.64278, [783] := 47.408234, [784] := 56.44969, [785] := 64.953415, [786] := 73.06321, [787] := 79.04708, [788] := 85.85005, [789] := 91.64634, [790] := 96.26086, [791] := 99.32471, [792] := 100.68154, [793] := 101.10673, [794] := 100.3564, [795] := 98.50559, [796] := 96.42968, [797] := 93.14075, [798] := 88.957664, [799] := 84.349396, [800] := 84.349396);
   VPotencia : REAL[1500] := ([0] := 5.9449345e-37, [1] := 5.9449345e-37, [2] := 5.9449345e-37, [3] := 5.9449345e-37, [4] := 5.9449345e-37, [5] := 5.9449345e-37, [6] := 5.9449345e-37, [7] := 5.9449345e-37, [8] := 5.9449345e-37, [9] := 5.9449345e-37, [10] := 5.9449345e-37, [11] := 5.9449345e-37, [12] := 5.9449345e-37, [13] := 5.9449345e-37, [14] := 5.9449345e-37, [15] := 5.9449345e-37, [16] := 5.9449345e-37, [17] := 5.9449345e-37, [18] := 5.9449345e-37, [19] := 5.9449345e-37, [20] := 5.9449345e-37, [21] := 5.9449345e-37, [22] := 5.9449345e-37, [23] := 5.9449345e-37, [24] := 5.9449345e-37, [25] := 5.9449345e-37, [26] := 5.9449345e-37, [27] := 5.9449345e-37, [28] := 5.9449345e-37, [29] := 5.9449345e-37, [30] := 5.9449345e-37, [31] := 5.9449345e-37, [32] := 5.9449345e-37, [33] := 5.9449345e-37, [34] := 5.9449345e-37, [35] := 5.9449345e-37, [36] := 5.9449345e-37, [37] := 5.9449345e-37, [38] := 5.9449345e-37, [39] := 5.9449345e-37, [40] := 5.9449345e-37, [41] := 5.9449345e-37, [42] := 5.9449345e-37, [43] := 5.9449345e-37, [44] := 5.9449345e-37, [45] := 5.9449345e-37, [46] := 5.9449345e-37, [47] := 5.9449345e-37, [48] := 5.9449345e-37, [49] := 5.9449345e-37, [50] := 5.9449345e-37, [51] := 5.9449345e-37, [52] := 5.9449345e-37, [53] := 5.9449345e-37, [54] := 5.9449345e-37, [55] := 5.9449345e-37, [56] := 5.9449345e-37, [57] := 5.9449345e-37, [58] := 5.9449345e-37, [59] := 5.9449345e-37,
        [60] := 5.9449345e-37, [61] := 5.9449345e-37, [62] := 5.9449345e-37, [63] := 5.9449345e-37, [64] := 5.9449345e-37, [65] := 5.9449345e-37, [66] := 5.9449345e-37, [67] := 5.9449345e-37, [68] := 5.9449345e-37, [69] := 5.9449345e-37, [70] := 5.9449345e-37, [71] := 5.9449345e-37, [72] := 5.9449345e-37, [73] := 5.9449345e-37, [74] := 5.9449345e-37, [75] := 5.9449345e-37, [76] := 5.9449345e-37, [77] := 5.9449345e-37, [78] := 5.9449345e-37, [79] := 5.9449345e-37, [80] := 5.9449345e-37, [81] := 5.9449345e-37, [82] := 5.9449345e-37, [83] := 5.9449345e-37, [84] := 5.9449345e-37, [85] := 5.9449345e-37, [86] := 5.9449345e-37, [87] := 5.9449345e-37, [88] := 5.9449345e-37, [89] := 5.9449345e-37, [90] := 5.9449345e-37, [91] := 5.9449345e-37, [92] := 5.9449345e-37, [93] := 5.9449345e-37, [94] := 5.9449345e-37, [95] := 5.9449345e-37, [96] := 5.9449345e-37, [97] := 5.9449345e-37, [98] := 5.9449345e-37, [99] := 5.9449345e-37, [100] := 5.9449345e-37, [101] := 5.9449345e-37, [102] := 5.9449345e-37, [103] := 5.9449345e-37, [104] := 5.9449345e-37, [105] := 5.9449345e-37, [106] := 5.9449345e-37, [107] := 5.9449345e-37, [108] := 5.9449345e-37, [109] := 5.9449345e-37, [110] := 5.9449345e-37, [111] := 5.9449345e-37, [112] := 5.9449345e-37, [113] := 5.9449345e-37, [114] := 5.9449345e-37, [115] := 5.9449345e-37, [116] := 5.9449345e-37, [117] := 5.9449345e-37, [118] := 5.9449345e-37, [119] := 5.9449345e-37,
        [120] := 5.9449345e-37, [121] := 5.9449345e-37, [122] := 5.9449345e-37, [123] := 5.9449345e-37, [124] := 5.9449345e-37, [125] := 5.9449345e-37, [126] := 5.9449345e-37, [127] := 5.9449345e-37, [128] := 5.9449345e-37, [129] := 5.9449345e-37, [130] := 5.9449345e-37, [131] := 5.9449345e-37, [132] := 5.9449345e-37, [133] := 5.9449345e-37, [134] := 5.9449345e-37, [135] := 5.9449345e-37, [136] := 5.9449345e-37, [137] := 5.9449345e-37, [138] := 5.9449345e-37, [139] := 5.9449345e-37, [140] := 5.9449345e-37, [141] := 5.9449345e-37, [142] := 5.9449345e-37, [143] := 5.9449345e-37, [144] := 5.9449345e-37, [145] := 5.9449345e-37, [146] := 5.9449345e-37, [147] := 5.9449345e-37, [148] := 5.9449345e-37, [149] := 5.9449345e-37, [150] := 5.9449345e-37, [151] := 5.9449345e-37, [152] := 5.9449345e-37, [153] := 5.9449345e-37, [154] := 5.9449345e-37, [155] := 5.9449345e-37, [156] := 5.9449345e-37, [157] := 5.9449345e-37, [158] := 5.9449345e-37, [159] := 5.9449345e-37, [160] := 5.9449345e-37, [161] := 5.9449345e-37, [162] := 5.9449345e-37, [163] := 5.9449345e-37, [164] := 5.9449345e-37, [165] := 5.9449345e-37, [166] := 5.9449345e-37, [167] := 5.9449345e-37, [168] := 5.9449345e-37, [169] := 5.9449345e-37, [170] := 5.9449345e-37, [171] := 5.9449345e-37, [172] := 5.9449345e-37, [173] := 5.9449345e-37, [174] := 5.9449345e-37, [175] := 5.9449345e-37, [176] := 5.9449345e-37, [177] := 5.9449345e-37, [178] := 5.9449345e-37, [179] := 5.9449345e-37,
        [180] := 5.9449345e-37, [181] := 5.9449345e-37, [182] := 5.9449345e-37, [183] := 5.9449345e-37, [184] := 5.9449345e-37, [185] := 5.9449345e-37, [186] := 5.9449345e-37, [187] := 5.9449345e-37, [188] := 5.9449345e-37, [189] := 5.9449345e-37, [190] := 5.9449345e-37, [191] := 5.9449345e-37, [192] := 5.9449345e-37, [193] := 5.9449345e-37, [194] := 5.9449345e-37, [195] := 5.9449345e-37, [196] := 5.9449345e-37, [197] := 5.9449345e-37, [198] := 5.9449345e-37, [199] := 5.9449345e-37, [200] := 5.9449345e-37, [201] := 5.9449345e-37, [202] := 5.9449345e-37, [203] := 5.9449345e-37, [204] := 5.9449345e-37, [205] := 5.9449345e-37, [206] := 5.9449345e-37, [207] := 5.9449345e-37, [208] := 5.9449345e-37, [209] := 5.9449345e-37, [210] := 5.9449345e-37, [211] := 5.9449345e-37, [212] := 5.9449345e-37, [213] := 5.9449345e-37, [214] := 5.9449345e-37, [215] := 5.9449345e-37, [216] := 5.9449345e-37, [217] := 5.9449345e-37, [218] := 5.9449345e-37, [219] := 5.9449345e-37, [220] := 5.9449345e-37, [221] := 5.9449345e-37, [222] := 5.9449345e-37, [223] := 5.9449345e-37, [224] := 5.9449345e-37, [225] := 5.9449345e-37, [226] := 5.9449345e-37, [227] := 5.9449345e-37, [228] := 5.9449345e-37, [229] := 5.9449345e-37, [230] := 5.9449345e-37, [231] := 5.9449345e-37, [232] := 5.9449345e-37, [233] := 5.9449345e-37, [234] := 5.9449345e-37, [235] := 5.9449345e-37, [236] := 5.9449345e-37, [237] := 5.9449345e-37, [238] := 5.9449345e-37, [239] := 5.9449345e-37,
        [240] := 5.9449345e-37, [241] := 5.9449345e-37, [242] := 5.9449345e-37, [243] := 5.9449345e-37, [244] := 5.9449345e-37, [245] := 5.9449345e-37, [246] := 5.9449345e-37, [247] := 5.9449345e-37, [248] := 5.9449345e-37, [249] := 5.9449345e-37, [250] := 5.9449345e-37, [251] := 5.9449345e-37, [252] := 5.9449345e-37, [253] := 5.9449345e-37, [254] := 5.9449345e-37, [255] := 5.9449345e-37, [256] := 5.9449345e-37, [257] := 5.9449345e-37, [258] := 5.9449345e-37, [259] := 5.9449345e-37, [260] := 5.9449345e-37, [261] := 5.9449345e-37, [262] := 5.9449345e-37, [263] := 5.9449345e-37, [264] := 5.9449345e-37, [265] := 5.9449345e-37, [266] := 5.9449345e-37, [267] := 5.9449345e-37, [268] := 5.9449345e-37, [269] := 5.9449345e-37, [270] := 5.9449345e-37, [271] := 5.9449345e-37, [272] := 5.9449345e-37, [273] := 5.9449345e-37, [274] := 5.9449345e-37, [275] := 5.9449345e-37, [276] := 5.9449345e-37, [277] := 5.9449345e-37, [278] := 5.9449345e-37, [279] := 5.9449345e-37, [280] := 5.9449345e-37, [281] := 5.9449345e-37, [282] := 5.9449345e-37, [283] := 5.9449345e-37, [284] := 5.9449345e-37, [285] := 5.9449345e-37, [286] := 5.9449345e-37, [287] := 5.9449345e-37, [288] := 5.9449345e-37, [289] := 5.9449345e-37, [290] := 5.9449345e-37, [291] := 5.9449345e-37, [292] := 5.9449345e-37, [293] := 5.9449345e-37, [294] := 5.9449345e-37, [295] := 5.9449345e-37, [296] := 5.9449345e-37, [297] := 5.9449345e-37, [298] := 5.9449345e-37, [299] := 5.9449345e-37,
        [300] := 5.9449345e-37, [301] := 5.9449345e-37, [302] := 5.9449345e-37, [303] := 5.9449345e-37, [304] := 5.9449345e-37, [305] := 5.9449345e-37, [306] := 5.9449345e-37, [307] := 5.9449345e-37, [308] := 5.9449345e-37, [309] := 5.9449345e-37, [310] := 5.9449345e-37, [311] := 5.9449345e-37, [312] := 5.9449345e-37, [313] := 5.9449345e-37, [314] := 5.9449345e-37, [315] := 5.9449345e-37, [316] := 5.9449345e-37, [317] := 5.9449345e-37, [318] := 5.9449345e-37, [319] := 5.9449345e-37, [320] := 5.9449345e-37, [321] := 5.9449345e-37, [322] := 5.9449345e-37, [323] := 5.9449345e-37, [324] := 5.9449345e-37, [325] := 5.9449345e-37, [326] := 5.9449345e-37, [327] := 5.9449345e-37, [328] := 5.9449345e-37, [329] := 5.9449345e-37, [330] := 5.9449345e-37, [331] := 5.9449345e-37, [332] := 5.9449345e-37, [333] := 5.9449345e-37, [334] := 5.9449345e-37, [335] := 5.9449345e-37, [336] := 5.9449345e-37, [337] := 5.9449345e-37, [338] := 5.9449345e-37, [339] := 5.9449345e-37, [340] := 5.9449345e-37, [341] := 5.9449345e-37, [342] := 5.9449345e-37, [343] := 5.9449345e-37, [344] := 5.9449345e-37, [345] := 5.9449345e-37, [346] := 5.9449345e-37, [347] := 5.9449345e-37, [348] := 5.9449345e-37, [349] := 5.9449345e-37, [350] := 5.9449345e-37, [351] := 5.9449345e-37, [352] := 5.9449345e-37, [353] := 5.9449345e-37, [354] := 5.9449345e-37, [355] := 5.9449345e-37, [356] := 5.9449345e-37, [357] := 5.9449345e-37, [358] := 5.9449345e-37, [359] := 5.9449345e-37,
        [360] := 5.9449345e-37, [361] := 5.9449345e-37, [362] := 5.9449345e-37, [363] := 5.9449345e-37, [364] := 5.9449345e-37, [365] := 5.9449345e-37, [366] := 5.9449345e-37, [367] := 5.9449345e-37, [368] := 5.9449345e-37, [369] := 5.9449345e-37, [370] := 5.9449345e-37, [371] := 5.9449345e-37, [372] := 5.9449345e-37, [373] := 5.9449345e-37, [374] := 5.9449345e-37, [375] := 5.9449345e-37, [376] := 5.9449345e-37, [377] := 5.9449345e-37, [378] := 5.9449345e-37, [379] := 5.9449345e-37, [380] := 5.9449345e-37, [381] := 5.9449345e-37, [382] := 5.9449345e-37, [383] := 5.9449345e-37, [384] := 5.9449345e-37, [385] := 5.9449345e-37, [386] := 5.9449345e-37, [387] := 5.9449345e-37, [388] := 5.9449345e-37, [389] := 5.9449345e-37, [390] := 5.9449345e-37, [391] := 5.9449345e-37, [392] := 5.9449345e-37, [393] := 5.9449345e-37, [394] := 5.9449345e-37, [395] := 5.9449345e-37, [396] := 5.9449345e-37, [397] := 5.9449345e-37, [398] := 5.9449345e-37, [399] := 5.9449345e-37, [400] := 5.9449345e-37, [401] := 5.9449345e-37, [402] := 5.9449345e-37, [403] := 5.9449345e-37, [404] := 5.9449345e-37, [405] := 5.9449345e-37, [406] := 5.9449345e-37, [407] := 5.9449345e-37, [408] := 5.9449345e-37, [409] := 5.9449345e-37, [410] := 5.9449345e-37, [411] := 5.9449345e-37, [412] := 5.9449345e-37, [413] := 5.9449345e-37, [414] := 5.9449345e-37, [415] := 5.9449345e-37, [416] := 5.9449345e-37, [417] := 5.9449345e-37, [418] := 5.9449345e-37, [419] := 5.9449345e-37,
        [420] := 5.9449345e-37, [421] := 5.9449345e-37, [422] := 5.9449345e-37, [423] := 5.9449345e-37, [424] := 5.9449345e-37, [425] := 5.9449345e-37, [426] := 5.9449345e-37, [427] := 5.9449345e-37, [428] := 5.9449345e-37, [429] := 5.9449345e-37, [430] := 5.9449345e-37, [431] := 5.9449345e-37, [432] := 5.9449345e-37, [433] := 5.9449345e-37, [434] := 5.9449345e-37, [435] := 5.9449345e-37, [436] := 5.9449345e-37, [437] := 5.9449345e-37, [438] := 5.9449345e-37, [439] := 5.9449345e-37, [440] := 5.9449345e-37, [441] := 5.9449345e-37, [442] := 5.9449345e-37, [443] := 5.9449345e-37, [444] := 5.9449345e-37, [445] := 5.9449345e-37, [446] := 5.9449345e-37, [447] := 5.9449345e-37, [448] := 5.9449345e-37, [449] := 5.9449345e-37, [450] := 5.9449345e-37, [451] := 5.9449345e-37, [452] := 5.9449345e-37, [453] := 5.9449345e-37, [454] := 5.9449345e-37, [455] := 5.9449345e-37, [456] := 5.9449345e-37, [457] := 5.9449345e-37, [458] := 5.9449345e-37, [459] := 5.9449345e-37, [460] := 5.9449345e-37, [461] := 5.9449345e-37, [462] := 5.9449345e-37, [463] := 5.9449345e-37, [464] := 5.9449345e-37, [465] := 5.9449345e-37, [466] := 5.9449345e-37, [467] := 5.9449345e-37, [468] := 5.9449345e-37, [469] := 5.9449345e-37, [470] := 5.9449345e-37, [471] := 5.9449345e-37, [472] := 5.9449345e-37, [473] := 5.9449345e-37, [474] := 5.9449345e-37, [475] := 5.9449345e-37, [476] := 5.9449345e-37, [477] := 5.9449345e-37, [478] := 5.9449345e-37, [479] := 5.9449345e-37,
        [480] := 5.9449345e-37, [481] := 5.9449345e-37, [482] := 5.9449345e-37, [483] := 5.9449345e-37, [484] := 5.9449345e-37, [485] := 5.9449345e-37, [486] := 5.9449345e-37, [487] := 5.9449345e-37, [488] := 5.9449345e-37, [489] := 5.9449345e-37, [490] := 5.9449345e-37, [491] := 5.9449345e-37, [492] := 5.9449345e-37, [493] := 5.9449345e-37, [494] := 5.9449345e-37, [495] := 5.9449345e-37, [496] := 5.9449345e-37, [497] := 5.9449345e-37, [498] := 5.9449345e-37, [499] := 5.9449345e-37, [500] := 5.9449345e-37, [501] := 5.9449345e-37, [502] := 5.9449345e-37, [503] := 5.9449345e-37, [504] := 5.9449345e-37, [505] := 5.9449345e-37, [506] := 5.9449345e-37, [507] := 5.9449345e-37, [508] := 5.9449345e-37, [509] := 5.9449345e-37, [510] := 5.9449345e-37, [511] := 5.9449345e-37, [512] := 5.9449345e-37, [513] := 5.9449345e-37, [514] := 5.9449345e-37, [515] := 5.9449345e-37, [516] := 5.9449345e-37, [517] := 5.9449345e-37, [518] := 5.9449345e-37, [519] := 5.9449345e-37, [520] := 5.9449345e-37, [521] := 5.9449345e-37, [522] := 5.9449345e-37, [523] := 5.9449345e-37, [524] := 5.9449345e-37, [525] := 5.9449345e-37, [526] := 5.9449345e-37, [527] := 5.9449345e-37, [528] := 5.9449345e-37, [529] := 5.9449345e-37, [530] := 5.9449345e-37, [531] := 5.9449345e-37, [532] := 5.9449345e-37, [533] := 5.9449345e-37, [534] := 5.9449345e-37, [535] := 5.9449345e-37, [536] := 5.9449345e-37, [537] := 5.9449345e-37, [538] := 5.9449345e-37, [539] := 5.9449345e-37,
        [540] := 5.9449345e-37, [541] := 5.9449345e-37, [542] := 5.9449345e-37, [543] := 5.9449345e-37, [544] := 5.9449345e-37, [545] := 5.9449345e-37, [546] := 5.9449345e-37, [547] := 5.9449345e-37, [548] := 5.9449345e-37, [549] := 5.9449345e-37, [550] := 5.9449345e-37, [551] := 5.9449345e-37, [552] := 5.9449345e-37, [553] := 5.9449345e-37, [554] := 5.9449345e-37, [555] := 5.9449345e-37, [556] := 5.9449345e-37, [557] := 5.9449345e-37, [558] := 5.9449345e-37, [559] := 5.9449345e-37, [560] := 5.9449345e-37, [561] := 5.9449345e-37, [562] := 5.9449345e-37, [563] := 5.9449345e-37, [564] := 5.9449345e-37, [565] := 5.9449345e-37, [566] := 5.9449345e-37, [567] := 5.9449345e-37, [568] := 5.9449345e-37, [569] := 5.9449345e-37, [570] := 5.9449345e-37, [571] := 5.9449345e-37, [572] := 5.9449345e-37, [573] := 5.9449345e-37, [574] := 5.9449345e-37, [575] := 5.9449345e-37, [576] := 5.9449345e-37, [577] := 5.9449345e-37, [578] := 5.9449345e-37, [579] := 5.9449345e-37, [580] := 5.9449345e-37, [581] := 5.9449345e-37, [582] := 5.9449345e-37, [583] := 5.9449345e-37, [584] := 5.9449345e-37, [585] := 5.9449345e-37, [586] := 5.9449345e-37, [587] := 5.9449345e-37, [588] := 5.9449345e-37, [589] := 5.9449345e-37, [590] := 5.9449345e-37, [591] := 5.9449345e-37, [592] := 5.9449345e-37, [593] := 5.9449345e-37, [594] := 5.9449345e-37, [595] := 5.9449345e-37, [596] := 5.9449345e-37, [597] := 5.9449345e-37, [598] := 5.9449345e-37, [599] := 5.9449345e-37,
        [600] := 5.9449345e-37, [601] := 5.9449345e-37, [602] := 5.9449345e-37, [603] := 5.9449345e-37, [604] := 5.9449345e-37, [605] := 5.9449345e-37, [606] := 5.9449345e-37, [607] := 5.9449345e-37, [608] := 5.9449345e-37, [609] := 5.9449345e-37, [610] := 5.9449345e-37, [611] := 5.9449345e-37, [612] := 5.9449345e-37, [613] := 5.9449345e-37, [614] := 5.9449345e-37, [615] := 5.9449345e-37, [616] := 5.9449345e-37, [617] := 5.9449345e-37, [618] := 5.9449345e-37, [619] := 5.9449345e-37, [620] := 5.9449345e-37, [621] := 5.9449345e-37, [622] := 5.9449345e-37, [623] := 5.9449345e-37, [624] := 5.9449345e-37, [625] := 5.9449345e-37, [626] := 5.9449345e-37, [627] := 5.9449345e-37, [628] := 5.9449345e-37, [629] := 5.9449345e-37, [630] := 5.9449345e-37, [631] := 5.9449345e-37, [632] := 5.9449345e-37, [633] := 5.9449345e-37, [634] := 5.9449345e-37, [635] := 5.9449345e-37, [636] := 5.9449345e-37, [637] := 5.9449345e-37, [638] := 5.9449345e-37, [639] := 5.9449345e-37, [640] := 5.9449345e-37, [641] := 5.9449345e-37, [642] := 5.9449345e-37, [643] := 5.9449345e-37, [644] := 5.9449345e-37, [645] := 5.9449345e-37, [646] := 5.9449345e-37, [647] := 5.9449345e-37, [648] := 5.9449345e-37, [649] := 5.9449345e-37, [650] := 5.9449345e-37, [651] := 5.9449345e-37, [652] := 5.9449345e-37, [653] := 5.9449345e-37, [654] := 5.9449345e-37, [655] := 5.9449345e-37, [656] := 5.9449345e-37, [657] := 5.9449345e-37, [658] := 5.9449345e-37, [659] := 5.9449345e-37,
        [660] := 5.9449345e-37, [661] := 5.9449345e-37, [662] := 5.9449345e-37, [663] := 5.9449345e-37, [664] := 5.9449345e-37, [665] := 5.9449345e-37, [666] := 5.9449345e-37, [667] := 5.9449345e-37, [668] := 5.9449345e-37, [669] := 5.9449345e-37, [670] := 5.9449345e-37, [671] := 5.9449345e-37, [672] := 5.9449345e-37, [673] := 5.9449345e-37, [674] := 5.9449345e-37, [675] := 5.9449345e-37, [676] := 5.9449345e-37, [677] := 5.9449345e-37, [678] := 5.9449345e-37, [679] := 5.9449345e-37, [680] := 5.9449345e-37, [681] := 5.9449345e-37, [682] := 5.9449345e-37, [683] := 5.9449345e-37, [684] := 5.9449345e-37, [685] := 5.9449345e-37, [686] := 5.9449345e-37, [687] := 5.9449345e-37, [688] := 5.9449345e-37, [689] := 5.9449345e-37, [690] := 5.9449345e-37, [691] := 5.9449345e-37, [692] := 5.9449345e-37, [693] := 5.9449345e-37, [694] := 5.9449345e-37, [695] := 5.9449345e-37, [696] := 5.9449345e-37, [697] := 5.9449345e-37, [698] := 5.9449345e-37, [699] := 5.9449345e-37, [700] := 5.9449345e-37, [701] := 5.9449345e-37, [702] := 5.9449345e-37, [703] := 5.9449345e-37, [704] := 5.9449345e-37, [705] := 5.9449345e-37, [706] := 5.9449345e-37, [707] := 5.9449345e-37, [708] := 5.9449345e-37, [709] := 5.9449345e-37, [710] := 5.9449345e-37, [711] := 5.9449345e-37, [712] := 5.9449345e-37, [713] := 5.9449345e-37, [714] := 5.9449345e-37, [715] := 5.9449345e-37, [716] := 5.9449345e-37, [717] := 5.9449345e-37, [718] := 5.9449345e-37, [719] := 5.9449345e-37,
        [720] := 5.9449345e-37, [721] := 5.9449345e-37, [722] := 5.9449345e-37, [723] := 5.9449345e-37, [724] := 5.9449345e-37, [725] := 5.9449345e-37, [726] := 5.9449345e-37, [727] := 5.9449345e-37, [728] := 5.9449345e-37, [729] := 5.9449345e-37, [730] := 5.9449345e-37, [731] := 5.9449345e-37, [732] := 5.9449345e-37, [733] := 5.9449345e-37, [734] := 5.9449345e-37, [735] := 5.9449345e-37, [736] := 5.9449345e-37, [737] := 5.9449345e-37, [738] := 5.9449345e-37, [739] := 5.9449345e-37, [740] := 5.9449345e-37, [741] := 5.9449345e-37, [742] := 5.9449345e-37, [743] := 5.9449345e-37, [744] := 5.9449345e-37, [745] := 5.9449345e-37, [746] := 5.9449345e-37, [747] := 5.9449345e-37, [748] := 5.9449345e-37, [749] := 5.9449345e-37, [750] := 5.9449345e-37, [751] := 5.9449345e-37, [752] := 5.9449345e-37, [753] := 5.9449345e-37, [754] := 5.9449345e-37, [755] := 5.9449345e-37, [756] := 5.9449345e-37, [757] := 5.9449345e-37, [758] := 5.9449345e-37, [759] := 5.9449345e-37, [760] := 5.9449345e-37, [761] := 5.9449345e-37, [762] := 5.9449345e-37, [763] := 5.9449345e-37, [764] := 5.9449345e-37, [765] := 5.9449345e-37, [766] := 5.9449345e-37, [767] := 5.9449345e-37, [768] := 5.9449345e-37, [769] := 5.9449345e-37, [770] := 5.9449345e-37, [771] := 5.9449345e-37, [772] := 5.9449345e-37, [773] := 5.9449345e-37, [774] := 5.9449345e-37, [775] := 5.9449345e-37, [776] := 5.9449345e-37, [777] := 5.9449345e-37, [778] := 5.9449345e-37, [779] := 5.9449345e-37,
        [780] := 5.9449345e-37, [781] := 5.9449345e-37, [782] := 5.9449345e-37, [783] := 5.9449345e-37, [784] := 5.9449345e-37, [785] := 5.9449345e-37, [786] := 5.9449345e-37, [787] := 5.9449345e-37, [788] := 5.9449345e-37, [789] := 5.9449345e-37, [790] := 5.9449345e-37, [791] := 5.9449345e-37, [792] := 5.9449345e-37, [793] := 5.9449345e-37, [794] := 5.9449345e-37, [795] := 5.9449345e-37, [796] := 5.9449345e-37, [797] := 5.9449345e-37, [798] := 5.9449345e-37, [799] := 5.9449345e-37, [800] := 5.9449345e-37);
   VProximetro : BOOL[1504];
END_VAR

ROUTINE R001_ABB_Drive   (* ladder *)
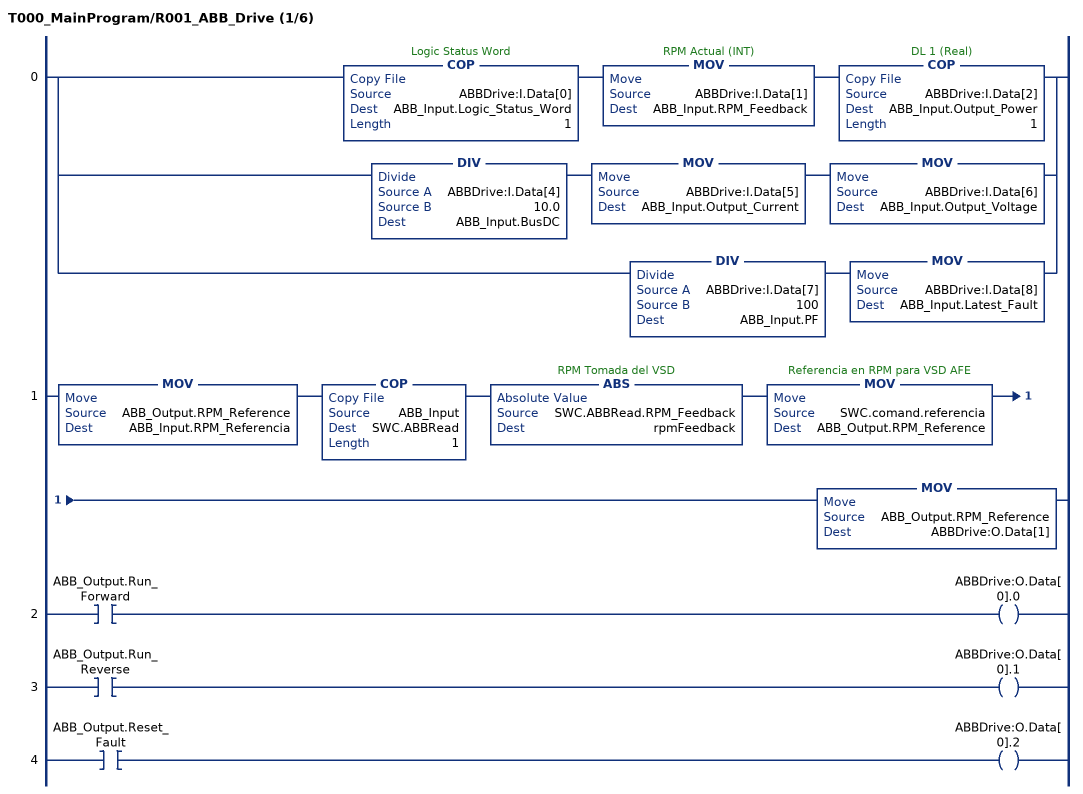
   0: [COP(ABBDrive:I.Data[0],ABB_Input.Logic_Status_Word,1) MOV(ABBDrive:I.Data[1],ABB_Input.RPM_Feedback) COP(ABBDrive:I.Data[2],ABB_Input.Output_Power,1) ,DIV(ABBDrive:I.Data[4],10.0,ABB_Input.BusDC) MOV(ABBDrive:I.Data[5],ABB_Input.Output_Current) MOV(ABBDrive:I.Data[6],ABB_Input.Output_Voltage) ,DIV(ABBDrive:I.Data[7],100,ABB_Input.PF) MOV(ABBDrive:I.Data[8],ABB_Input.Latest_Fault) ];
   1: MOV(ABB_Output.RPM_Reference,ABB_Input.RPM_Referencia)COP(ABB_Input,SWC.ABBRead,1)ABS(SWC.ABBRead.RPM_Feedback,rpmFeedback)MOV(SWC.comand.referencia,ABB_Output.RPM_Reference)MOV(ABB_Output.RPM_Reference,ABBDrive:O.Data[1]);
   2: XIC(ABB_Output.Run_Forward)OTE(ABBDrive:O.Data[0].0);
   3: XIC(ABB_Output.Run_Reverse)OTE(ABBDrive:O.Data[0].1);
   4: XIC(ABB_Output.Reset_Fault)OTE(ABBDrive:O.Data[0].2);
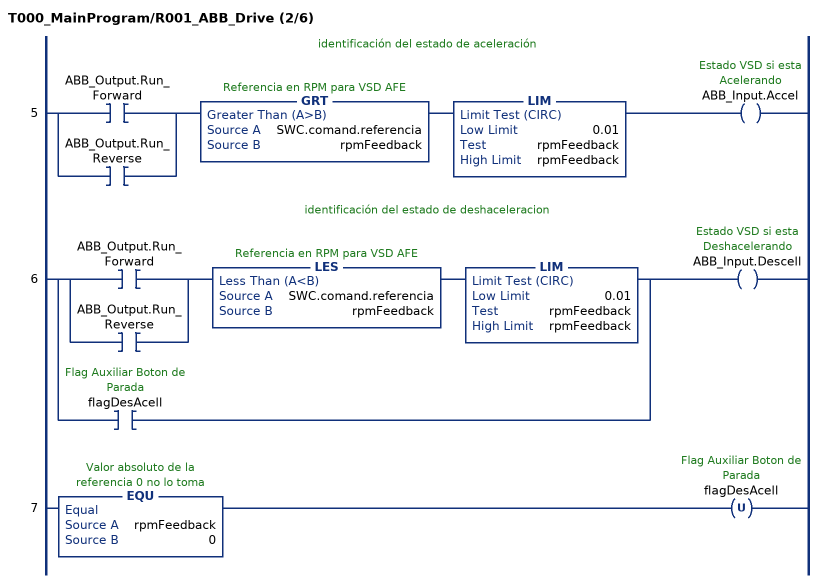
   // identificación del estado de aceleración
   5: [XIC(ABB_Output.Run_Forward) ,XIC(ABB_Output.Run_Reverse) ]GRT(SWC.comand.referencia,rpmFeedback)LIM(0.01,rpmFeedback,rpmFeedback)OTE(ABB_Input.Accel);
   // identificación del estado de deshaceleracion
   6: [[XIC(ABB_Output.Run_Forward) ,XIC(ABB_Output.Run_Reverse) ] LES(SWC.comand.referencia,rpmFeedback) LIM(0.01,rpmFeedback,rpmFeedback) ,XIC(flagDesAcell) ]OTE(ABB_Input.Descell);
   7: EQU(rpmFeedback,0)OTU(flagDesAcell);
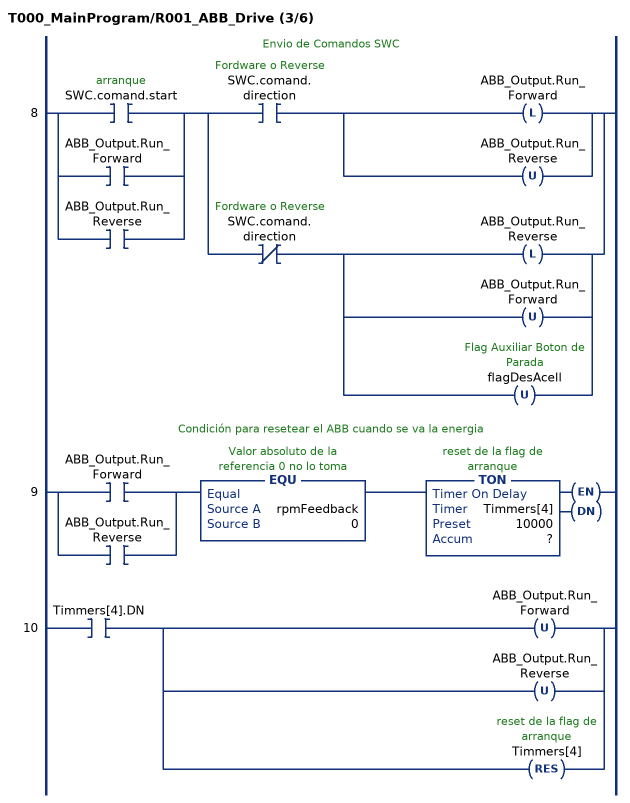
   // Envio de Comandos SWC
   8: [[XIC(SWC.comand.start) ,XIC(ABB_Output.Run_Forward) ] ,XIC(ABB_Output.Run_Reverse) ][XIC(SWC.comand.direction) [OTL(ABB_Output.Run_Forward) ,OTU(ABB_Output.Run_Reverse) ] ,XIO(SWC.comand.direction) [OTL(ABB_Output.Run_Reverse) ,[OTU(ABB_Output.Run_Forward) ,OTU(flagDesAcell) ] ] ];
   // Condición para resetear el ABB cuando se va la energia
   9: [XIC(ABB_Output.Run_Forward) ,XIC(ABB_Output.Run_Reverse) ]EQU(rpmFeedback,0)TON(Timmers[4],?,?);
   10: XIC(Timmers[4].DN)[OTU(ABB_Output.Run_Forward) ,[OTU(ABB_Output.Run_Reverse) ,RES(Timmers[4]) ] ];
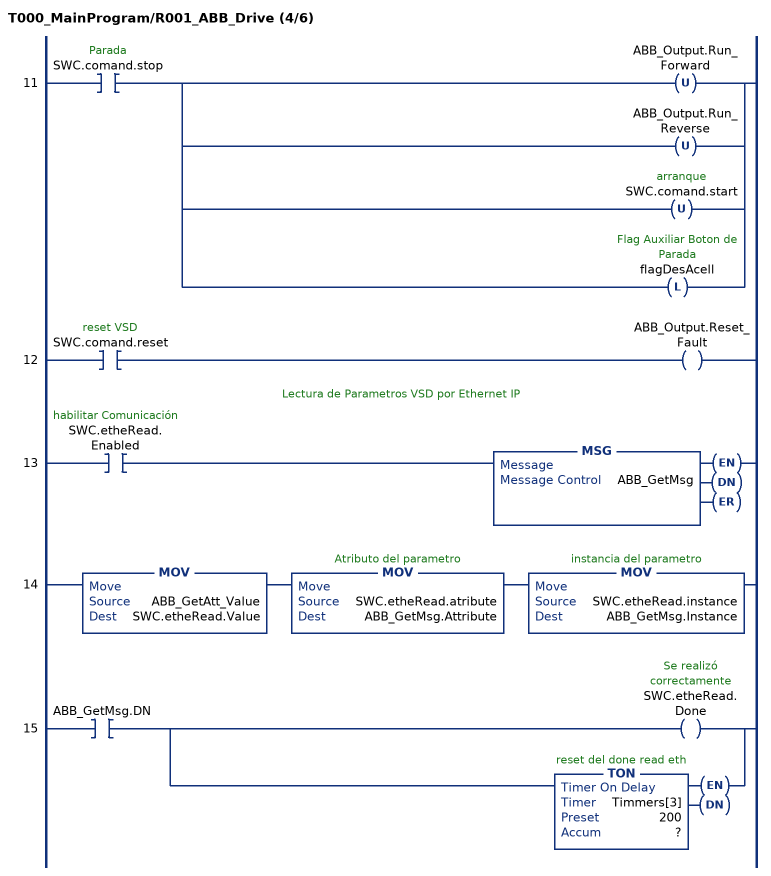
   11: XIC(SWC.comand.stop)[OTU(ABB_Output.Run_Forward) ,[OTU(ABB_Output.Run_Reverse) ,[OTU(SWC.comand.start) ,OTL(flagDesAcell) ] ] ];
   12: XIC(SWC.comand.reset)OTE(ABB_Output.Reset_Fault);
   // Lectura de Parametros VSD por Ethernet IP
   13: XIC(SWC.etheRead.Enabled)MSG(ABB_GetMsg);
   14: MOV(ABB_GetAtt_Value,SWC.etheRead.Value)MOV(SWC.etheRead.atribute,ABB_GetMsg.Attribute)MOV(SWC.etheRead.instance,ABB_GetMsg.Instance);
   15: XIC(ABB_GetMsg.DN)[OTE(SWC.etheRead.Done) ,TON(Timmers[3],?,?) ];
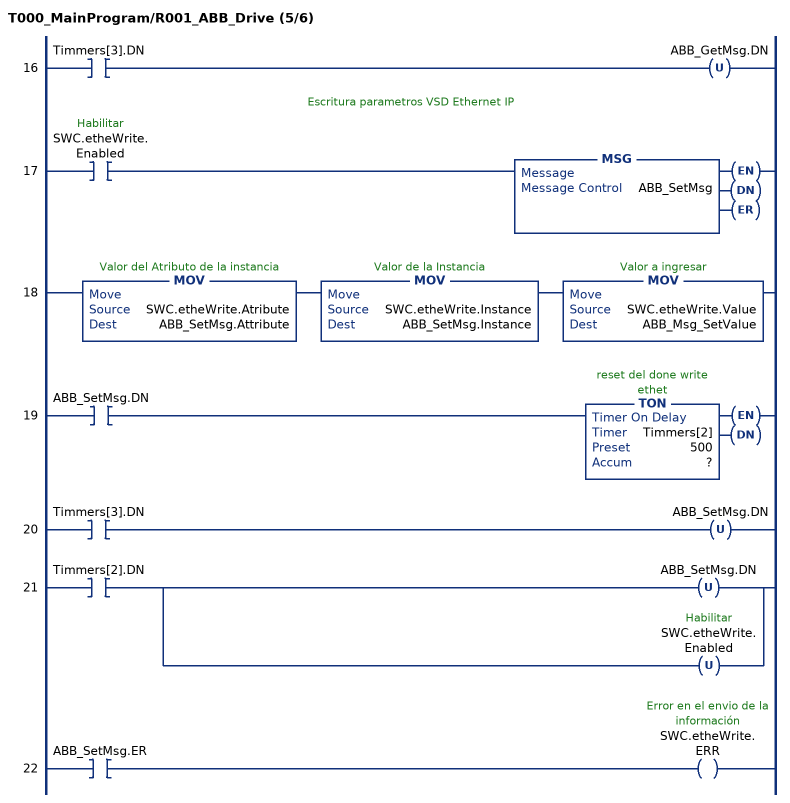
   16: XIC(Timmers[3].DN)OTU(ABB_GetMsg.DN);
   // Escritura parametros VSD Ethernet IP
   17: XIC(SWC.etheWrite.Enabled)MSG(ABB_SetMsg);
   18: MOV(SWC.etheWrite.Atribute,ABB_SetMsg.Attribute)MOV(SWC.etheWrite.Instance,ABB_SetMsg.Instance)MOV(SWC.etheWrite.Value,ABB_Msg_SetValue);
   19: XIC(ABB_SetMsg.DN)TON(Timmers[2],?,?);
   20: XIC(Timmers[3].DN)OTU(ABB_SetMsg.DN);
   21: XIC(Timmers[2].DN)[OTU(ABB_SetMsg.DN) ,OTU(SWC.etheWrite.Enabled) ];
   22: XIC(ABB_SetMsg.ER)OTE(SWC.etheWrite.ERR);
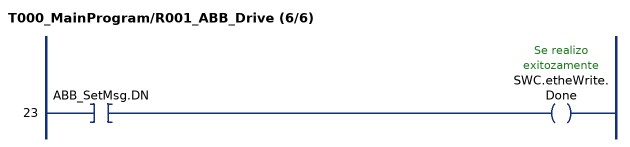
   23: XIC(ABB_SetMsg.DN)OTE(SWC.etheWrite.Done);
END_ROUTINE

ROUTINE R002_dinagramaPotencia   (* ladder *)
// Adquisión de los diferentes strokes para la captura del dinagrama de superficie
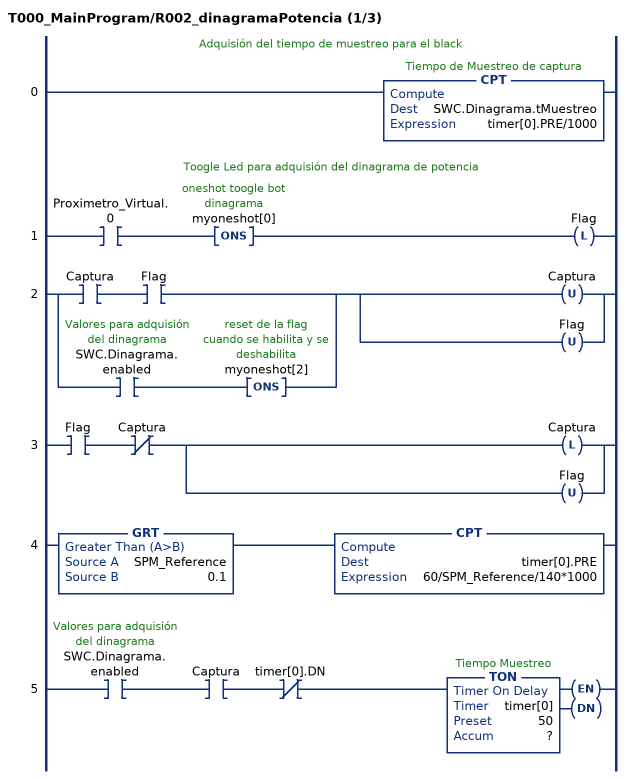
   // Adquisión del tiempo de muestreo para el black
   0: CPT(SWC.Dinagrama.tMuestreo,timer[0].PRE/1000);
   // Toogle Led para adquisión del dinagrama de potencia
   1: XIC(Proximetro_Virtual.0)ONS(myoneshot[0])OTL(Flag);
   2: [XIC(Captura) XIC(Flag) ,XIC(SWC.Dinagrama.enabled) ONS(myoneshot[2]) ][OTU(Captura) ,OTU(Flag) ];
   3: XIC(Flag)XIO(Captura)[OTL(Captura) ,OTU(Flag) ];
   4: GRT(SPM_Reference,0.1)CPT(timer[0].PRE,60/SPM_Reference/140*1000);
   5: XIC(SWC.Dinagrama.enabled)XIC(Captura)XIO(timer[0].DN)TON(timer[0],?,?);
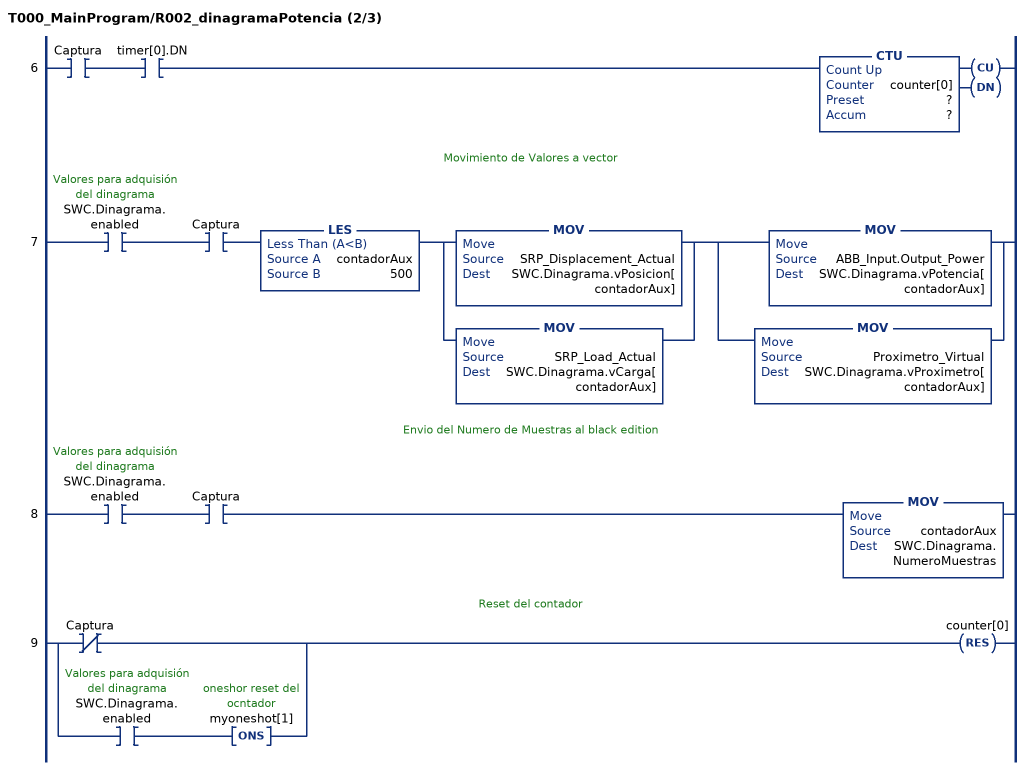
   6: XIC(Captura)XIC(timer[0].DN)CTU(counter[0],?,?);
   // Movimiento de Valores a vector
   7: XIC(SWC.Dinagrama.enabled)XIC(Captura)LES(contadorAux,500)[MOV(SRP_Displacement_Actual,SWC.Dinagrama.vPosicion[contadorAux]) ,MOV(SRP_Load_Actual,SWC.Dinagrama.vCarga[contadorAux]) ][MOV(ABB_Input.Output_Power,SWC.Dinagrama.vPotencia[contadorAux]) ,MOV(Proximetro_Virtual,SWC.Dinagrama.vProximetro[contadorAux]) ];
   // Envio del Numero de Muestras al black edition
   8: XIC(SWC.Dinagrama.enabled)XIC(Captura)MOV(contadorAux,SWC.Dinagrama.NumeroMuestras);
   // Reset del contador
   9: [XIO(Captura) ,XIC(SWC.Dinagrama.enabled) ONS(myoneshot[1]) ]RES(counter[0]);
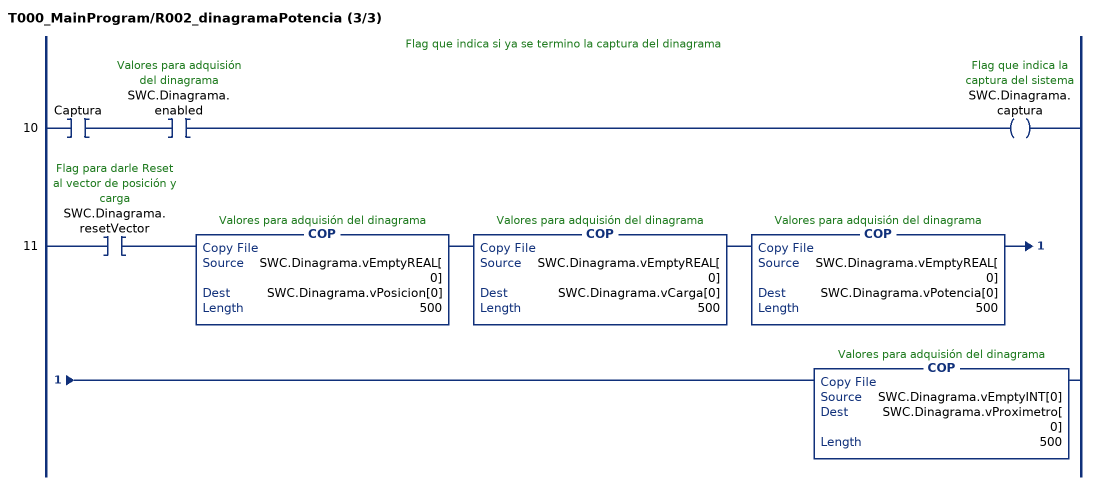
   // Flag que indica si ya se termino la captura del dinagrama
   10: XIC(Captura)XIC(SWC.Dinagrama.enabled)OTE(SWC.Dinagrama.captura);
   11: XIC(SWC.Dinagrama.resetVector)COP(SWC.Dinagrama.vEmptyREAL[0],SWC.Dinagrama.vPosicion[0],500)COP(SWC.Dinagrama.vEmptyREAL[0],SWC.Dinagrama.vCarga[0],500)COP(SWC.Dinagrama.vEmptyREAL[0],SWC.Dinagrama.vPotencia[0],500)COP(SWC.Dinagrama.vEmptyINT[0],SWC.Dinagrama.vProximetro[0],500);
END_ROUTINE

ROUTINE R003_IO_Digital   (* ladder *)
// Entradas Digitales
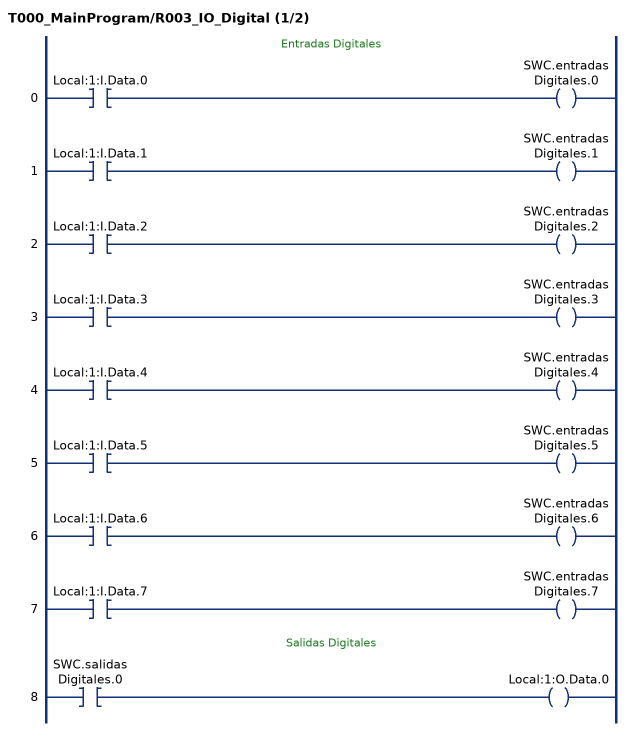
   // Entradas Digitales
   0: XIC(Local:1:I.Data.0)OTE(SWC.entradasDigitales.0);
   1: XIC(Local:1:I.Data.1)OTE(SWC.entradasDigitales.1);
   2: XIC(Local:1:I.Data.2)OTE(SWC.entradasDigitales.2);
   3: XIC(Local:1:I.Data.3)OTE(SWC.entradasDigitales.3);
   4: XIC(Local:1:I.Data.4)OTE(SWC.entradasDigitales.4);
   5: XIC(Local:1:I.Data.5)OTE(SWC.entradasDigitales.5);
   6: XIC(Local:1:I.Data.6)OTE(SWC.entradasDigitales.6);
   7: XIC(Local:1:I.Data.7)OTE(SWC.entradasDigitales.7);
   // Salidas Digitales
   8: XIC(SWC.salidasDigitales.0)OTE(Local:1:O.Data.0);
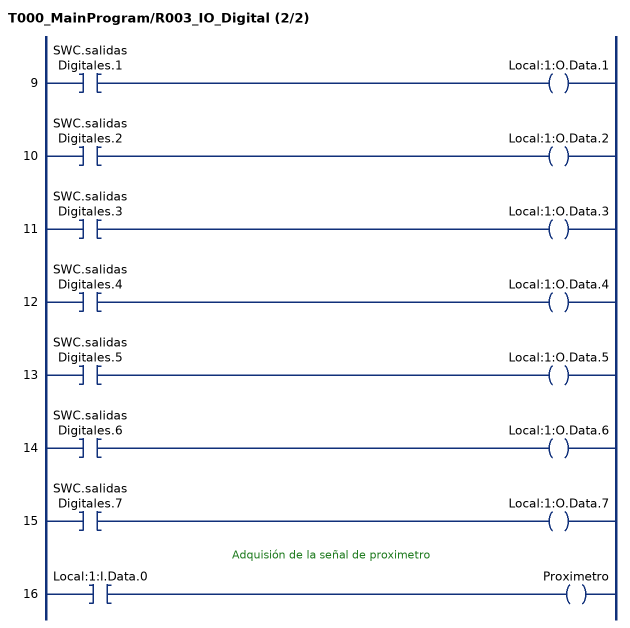
   9: XIC(SWC.salidasDigitales.1)OTE(Local:1:O.Data.1);
   10: XIC(SWC.salidasDigitales.2)OTE(Local:1:O.Data.2);
   11: XIC(SWC.salidasDigitales.3)OTE(Local:1:O.Data.3);
   12: XIC(SWC.salidasDigitales.4)OTE(Local:1:O.Data.4);
   13: XIC(SWC.salidasDigitales.5)OTE(Local:1:O.Data.5);
   14: XIC(SWC.salidasDigitales.6)OTE(Local:1:O.Data.6);
   15: XIC(SWC.salidasDigitales.7)OTE(Local:1:O.Data.7);
   // Adquisión de la señal de proximetro
   16: XIC(Local:1:I.Data.0)OTE(Proximetro);
END_ROUTINE

ROUTINE R004_IO_Anologica   (* function block diagram *)
// Rutina Para Entradas  Analogas
   SHEET 1
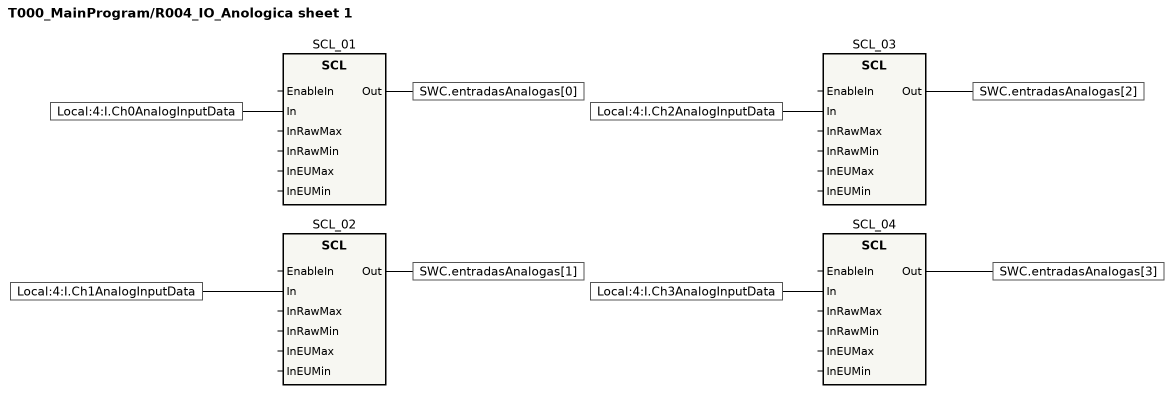
   SCL_01 : SCL(In := Local:4:I.Ch0AnalogInputData);   // unwired pins: EnableIn InRawMax InRawMin InEUMax InEUMin
   SCL_02 : SCL(In := Local:4:I.Ch1AnalogInputData);   // unwired pins: EnableIn InRawMax InRawMin InEUMax InEUMin
   SWC.entradasAnalogas[0] := SCL_01.Out;
   SWC.entradasAnalogas[1] := SCL_02.Out;
   SCL_03 : SCL(In := Local:4:I.Ch2AnalogInputData);   // unwired pins: EnableIn InRawMax InRawMin InEUMax InEUMin
   SCL_04 : SCL(In := Local:4:I.Ch3AnalogInputData);   // unwired pins: EnableIn InRawMax InRawMin InEUMax InEUMin
   SWC.entradasAnalogas[2] := SCL_03.Out;
   SWC.entradasAnalogas[3] := SCL_04.Out;
END_ROUTINE

ROUTINE R00_MainRoutine   (* ladder *)
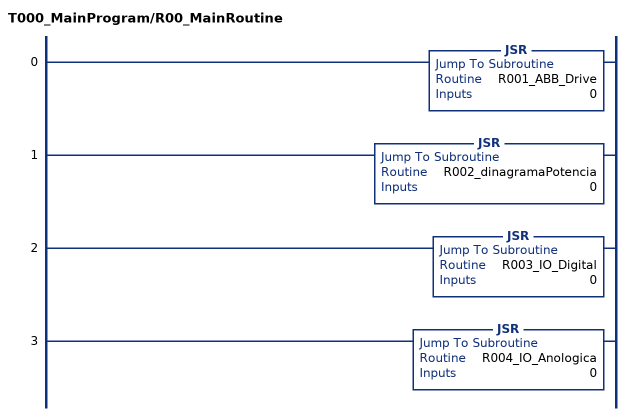
   0: JSR(R001_ABB_Drive,0);
   1: JSR(R002_dinagramaPotencia,0);
   2: JSR(R003_IO_Digital,0);
   3: JSR(R004_IO_Anologica,0);
END_ROUTINE
END_PROGRAM
